C01827=1144.684,360.117,-81.640,-176.368,9.412,148.862
C01828=1144.680,360.365,-81.675,-176.367,9.416,148.862
C01829=1144.676,360.613,-81.711,-176.364,9.420,148.863
C01830=1144.671,360.859,-81.746,-176.361,9.425,148.863
C01831=1144.667,361.107,-81.781,-176.358,9.429,148.863
C01832=1144.664,361.355,-81.817,-176.356,9.432,148.864
C01833=1144.660,361.602,-81.852,-176.353,9.436,148.864
C01834=1144.656,361.849,-81.888,-176.351,9.441,148.865
C01835=1144.652,362.097,-81.923,-176.348,9.445,148.865
C01836=1144.648,362.344,-81.959,-176.345,9.449,148.865
C01837=1144.644,362.592,-81.993,-176.344,9.453,148.866
C01838=1144.640,362.839,-82.029,-176.341,9.457,148.866
C01839=1144.637,363.087,-82.064,-176.338,9.461,148.866
C01840=1144.633,363.334,-82.100,-176.335,9.465,148.867
C01841=1144.629,363.582,-82.135,-176.333,9.470,148.867
C01842=1144.626,363.829,-82.171,-176.330,9.474,148.867
C01843=1144.621,364.077,-82.207,-176.328,9.477,148.868
C01844=1144.617,364.324,-82.242,-176.325,9.481,148.868
C01845=1144.613,364.571,-82.278,-176.322,9.486,148.869
C01846=1144.609,364.855,-82.318,-176.319,9.491,148.869
C01847=1144.604,365.138,-82.359,-176.316,9.495,148.869
C01848=1144.601,365.422,-82.400,-176.313,9.500,148.870
C01849=1144.596,365.705,-82.441,-176.310,9.504,148.870
C01850=1144.592,365.953,-82.477,-176.308,9.508,148.870
C01851=1144.587,366.200,-82.513,-176.305,9.513,148.871
C01852=1144.584,366.448,-82.548,-176.303,9.517,148.871
C01853=1144.580,366.695,-82.584,-176.300,9.521,148.872
C01854=1144.576,366.943,-82.620,-176.297,9.526,148.872
C01855=1144.572,367.190,-82.656,-176.294,9.530,148.872
C01856=1144.569,367.437,-82.692,-176.292,9.534,148.873
C01857=1144.565,367.685,-82.727,-176.289,9.538,148.873
C01858=1144.561,367.933,-82.763,-176.287,9.542,148.874
C01859=1144.556,368.179,-82.798,-176.284,9.546,148.874
C01860=1144.553,368.426,-82.835,-176.281,9.550,148.874
C01861=1144.549,368.674,-82.871,-176.279,9.555,148.875
C01862=1144.545,368.922,-82.906,-176.276,9.559,148.875
C01863=1144.542,369.168,-82.943,-176.273,9.563,148.875
C01864=1144.537,369.416,-82.979,-176.271,9.567,148.876
C01865=1144.534,369.664,-83.014,-176.268,9.572,148.876
C01866=1144.530,369.911,-83.051,-176.266,9.576,148.877
C01867=1144.526,370.158,-83.087,-176.263,9.580,148.877
C01868=1144.522,370.406,-83.122,-176.260,9.584,148.877
C01869=1144.518,370.653,-83.159,-176.258,9.588,148.878
C01870=1144.514,370.901,-83.195,-176.256,9.592,148.878
C01871=1144.511,371.148,-83.231,-176.253,9.596,148.879
C01872=1144.507,371.395,-83.267,-176.250,9.601,148.879
C01873=1144.503,371.643,-83.303,-176.248,9.605,148.879
C01874=1144.499,371.890,-83.340,-176.245,9.610,148.880
C01875=1144.495,372.138,-83.375,-176.243,9.614,148.880
C01876=1144.491,372.385,-83.412,-176.240,9.618,148.881
C01877=1144.487,372.632,-83.447,-176.238,9.622,148.881
C01878=1144.483,372.879,-83.484,-176.235,9.626,148.882
C01879=1144.480,373.126,-83.521,-176.233,9.630,148.882
C01880=1144.476,373.374,-83.557,-176.230,9.635,148.883
C01881=1144.472,373.621,-83.593,-176.228,9.639,148.883
C01882=1144.468,373.869,-83.629,-176.226,9.643,148.883
C01883=1144.465,374.116,-83.665,-176.223,9.647,148.884
C01884=1144.460,374.363,-83.702,-176.221,9.652,148.884
C01885=1144.457,374.610,-83.738,-176.218,9.656,148.885
C01886=1144.453,374.858,-83.775,-176.217,9.659,148.885
C01887=1144.449,375.105,-83.810,-176.214,9.664,148.886
C01888=1144.445,375.352,-83.847,-176.212,9.668,148.886
C01889=1144.441,375.599,-83.884,-176.210,9.672,148.887
C01890=1144.438,375.847,-83.921,-176.207,9.676,148.887
C01891=1144.434,376.095,-83.957,-176.205,9.681,148.888
C01892=1144.430,376.342,-83.993,-176.203,9.684,148.888
C01893=1144.426,376.589,-84.030,-176.201,9.689,148.889
C01894=1144.422,376.836,-84.067,-176.199,9.692,148.889
C01895=1144.418,377.084,-84.102,-176.197,9.697,148.890
C01896=1144.414,377.331,-84.139,-176.195,9.701,148.890
C01897=1144.410,377.578,-84.176,-176.193,9.705,148.891
C01898=1144.407,377.825,-84.212,-176.191,9.709,148.891
C01899=1144.403,378.073,-84.249,-176.189,9.713,148.892
C01900=1144.399,378.321,-84.286,-176.187,9.717,148.892
C01901=1144.396,378.567,-84.322,-176.185,9.721,148.893
C01902=1144.392,378.815,-84.359,-176.183,9.725,148.893
C01903=1144.387,379.062,-84.396,-176.181,9.729,148.894
C01904=1144.383,379.309,-84.432,-176.179,9.733,148.894
C01905=1144.380,379.556,-84.469,-176.178,9.737,148.895
C01906=1144.377,379.804,-84.506,-176.176,9.741,148.896
C01907=1144.372,380.051,-84.543,-176.175,9.745,148.896
C01908=1144.369,380.298,-84.579,-176.173,9.749,148.897
C01909=1144.365,380.545,-84.616,-176.171,9.752,148.897
C01910=1144.361,380.792,-84.653,-176.170,9.756,148.898
C01911=1144.357,381.039,-84.690,-176.168,9.760,148.898
C01912=1144.354,381.287,-84.726,-176.167,9.764,148.899
C01913=1144.350,381.534,-84.763,-176.166,9.767,148.900
C01914=1144.346,381.781,-84.800,-176.165,9.771,148.900
C01915=1144.342,382.029,-84.837,-176.163,9.775,148.901
C01916=1144.338,382.276,-84.874,-176.162,9.779,148.902
C01917=1144.335,382.523,-84.910,-176.161,9.782,148.902
C01918=1144.331,382.771,-84.947,-176.160,9.786,148.903
C01919=1144.327,383.018,-84.984,-176.159,9.789,148.904
C01920=1144.323,383.265,-85.021,-176.158,9.792,148.904
C01921=1144.319,383.512,-85.058,-176.157,9.796,148.905
C01922=1144.315,383.760,-85.095,-176.156,9.799,148.906
C01923=1144.312,384.007,-85.131,-176.156,9.803,148.906
C01924=1144.308,384.254,-85.168,-176.155,9.806,148.907
C01925=1144.304,384.501,-85.206,-176.154,9.809,148.908
C01926=1144.300,384.749,-85.243,-176.154,9.813,148.908
C01927=1144.296,384.996,-85.280,-176.153,9.816,148.909
C01928=1144.292,385.243,-85.317,-176.153,9.819,148.910
C01929=1144.289,385.490,-85.353,-176.152,9.823,148.911
C01930=1144.285,385.738,-85.390,-176.152,9.825,148.911
C01931=1144.281,385.984,-85.428,-176.152,9.829,148.912
C01932=1144.277,386.231,-85.465,-176.151,9.832,148.913
C01933=1144.273,386.479,-85.501,-176.151,9.835,148.914
C01934=1144.270,386.727,-85.539,-176.151,9.838,148.914
C01935=1144.266,386.974,-85.575,-176.151,9.841,148.915
C01936=1144.262,387.221,-85.612,-176.152,9.843,148.916
C01937=1144.259,387.467,-85.649,-176.151,9.847,148.917
C01938=1144.255,387.715,-85.687,-176.151,9.849,148.917
C01939=1144.251,387.962,-85.723,-176.151,9.852,148.918
C01940=1144.247,388.209,-85.760,-176.152,9.855,148.919
C01941=1144.243,388.456,-85.798,-176.152,9.857,148.920
C01942=1144.240,388.704,-85.835,-176.152,9.860,148.921
C01943=1144.235,388.951,-85.872,-176.152,9.863,148.921
C01944=1144.231,389.198,-85.909,-176.153,9.866,148.922
C01945=1144.228,389.446,-85.946,-176.153,9.868,148.923
C01946=1144.224,389.693,-85.984,-176.154,9.871,148.924
C01947=1144.221,389.940,-86.020,-176.154,9.874,148.924
C01948=1144.217,390.187,-86.057,-176.155,9.876,148.925
C01949=1144.213,390.435,-86.094,-176.155,9.879,148.926
C01950=1144.208,390.721,-86.138,-176.156,9.881,148.927
C01951=1144.205,391.009,-86.180,-176.156,9.884,148.928
C01952=1144.200,391.295,-86.224,-176.157,9.888,148.929
C01953=1144.195,391.582,-86.266,-176.158,9.890,148.930
C01954=1144.192,391.830,-86.304,-176.159,9.892,148.931
C01955=1144.188,392.076,-86.341,-176.160,9.895,148.932
C01956=1144.184,392.324,-86.378,-176.160,9.897,148.932
C01957=1144.180,392.571,-86.415,-176.161,9.899,148.933
C01958=1144.176,392.819,-86.452,-176.162,9.902,148.934
C01959=1144.173,393.065,-86.490,-176.163,9.904,148.935
C01960=1144.168,393.312,-86.526,-176.164,9.906,148.936
C01961=1144.165,393.560,-86.564,-176.164,9.909,148.937
C01962=1144.162,393.807,-86.601,-176.165,9.911,148.937
C01963=1144.158,394.054,-86.638,-176.166,9.913,148.938
C01964=1144.154,394.302,-86.675,-176.167,9.915,148.939
C01965=1144.150,394.549,-86.712,-176.168,9.918,148.940
C01966=1144.146,394.795,-86.749,-176.169,9.920,148.941
C01967=1144.142,395.043,-86.786,-176.170,9.922,148.941
C01968=1144.139,395.290,-86.823,-176.171,9.924,148.942
C01969=1144.135,395.538,-86.860,-176.172,9.926,148.943
C01970=1144.131,395.784,-86.898,-176.173,9.928,148.944
C01971=1144.127,396.032,-86.935,-176.174,9.930,148.945
C01972=1144.123,396.279,-86.972,-176.175,9.932,148.946
C01973=1144.120,396.526,-87.009,-176.177,9.934,148.946
C01974=1144.115,396.773,-87.046,-176.178,9.936,148.947
C01975=1144.112,397.021,-87.083,-176.179,9.938,148.948
C01976=1144.108,397.268,-87.121,-176.180,9.940,148.949
C01977=1144.104,397.515,-87.158,-176.181,9.942,148.950
C01978=1144.101,397.763,-87.195,-176.182,9.945,148.951
C01979=1144.096,398.010,-87.232,-176.183,9.947,148.951
C01980=1144.093,398.256,-87.270,-176.184,9.949,148.952
C01981=1144.089,398.504,-87.306,-176.185,9.951,148.953
C01982=1144.086,398.751,-87.343,-176.186,9.953,148.954
C01983=1144.082,398.998,-87.381,-176.187,9.955,148.955
C01984=1144.078,399.245,-87.417,-176.189,9.957,148.956
C01985=1144.074,399.493,-87.455,-176.190,9.959,148.956
C01986=1144.070,399.740,-87.492,-176.191,9.961,148.957
C01987=1144.067,399.987,-87.529,-176.193,9.963,148.958
C01988=1144.062,400.234,-87.566,-176.194,9.965,148.959
C01989=1144.059,400.482,-87.603,-176.195,9.967,148.960
C01990=1144.055,400.728,-87.641,-176.196,9.969,148.961
C01991=1144.051,400.975,-87.678,-176.197,9.971,148.962
C01992=1144.048,401.223,-87.715,-176.198,9.973,148.962
C01993=1144.044,401.470,-87.752,-176.199,9.975,148.963
C01994=1144.040,401.717,-87.789,-176.201,9.976,148.964
C01995=1144.036,401.964,-87.826,-176.202,9.978,148.965
C01996=1144.032,402.212,-87.863,-176.203,9.980,148.966
C01997=1144.028,402.459,-87.901,-176.204,9.982,148.967
C01998=1144.024,402.706,-87.938,-176.205,9.984,148.967
C01999=1144.021,402.954,-87.975,-176.206,9.986,148.968
C02000=1144.017,403.201,-88.012,-176.208,9.987,148.969
C02001=1144.013,403.448,-88.049,-176.209,9.990,148.970
C02002=1144.010,403.695,-88.086,-176.210,9.992,148.970
C02003=1144.006,403.942,-88.123,-176.211,9.994,148.971
C02004=1144.002,404.189,-88.161,-176.212,9.996,148.972
C02005=1143.998,404.436,-88.197,-176.213,9.998,148.973
C02006=1143.995,404.684,-88.235,-176.214,10.000,148.974
C02007=1143.991,404.931,-88.271,-176.216,10.001,148.975
C02008=1143.987,405.178,-88.309,-176.217,10.003,148.975
C02009=1143.983,405.426,-88.346,-176.218,10.005,148.976
C02010=1143.979,405.673,-88.383,-176.219,10.007,148.977
C02011=1143.975,405.919,-88.421,-176.220,10.009,148.978
C02012=1143.971,406.167,-88.458,-176.221,10.011,148.978
C02013=1143.968,406.414,-88.495,-176.222,10.013,148.979
C02014=1143.964,406.661,-88.532,-176.223,10.015,148.980
C02015=1143.960,406.908,-88.569,-176.224,10.017,148.981
C02016=1143.956,407.156,-88.606,-176.226,10.019,148.982
C02017=1143.952,407.403,-88.643,-176.227,10.021,148.983
C02018=1143.949,407.650,-88.681,-176.228,10.022,148.983
C02019=1143.944,407.897,-88.718,-176.229,10.024,148.984
C02020=1143.941,408.145,-88.755,-176.230,10.027,148.985
C02021=1143.938,408.391,-88.792,-176.231,10.029,148.986
C02022=1143.934,408.638,-88.829,-176.232,10.030,148.986
C02023=1143.930,408.886,-88.866,-176.233,10.032,148.987
C02024=1143.926,409.133,-88.903,-176.234,10.034,148.988
C02025=1143.922,409.380,-88.940,-176.235,10.037,148.989
C02026=1143.918,409.627,-88.977,-176.236,10.038,148.989
C02027=1143.915,409.875,-89.015,-176.237,10.040,148.990
C02028=1143.911,410.122,-89.052,-176.238,10.042,148.991
C02029=1143.907,410.369,-89.089,-176.239,10.044,148.992
C02030=1143.903,410.617,-89.126,-176.239,10.046,148.993
C02031=1143.899,410.864,-89.163,-176.241,10.048,148.993
C02032=1143.896,411.111,-89.201,-176.242,10.050,148.994
C02033=1143.892,411.358,-89.237,-176.242,10.052,148.995
C02034=1143.888,411.606,-89.275,-176.243,10.054,148.996
C02035=1143.884,411.852,-89.312,-176.243,10.057,148.996
C02036=1143.880,412.099,-89.349,-176.245,10.059,148.997
C02037=1143.877,412.347,-89.386,-176.246,10.061,148.998
C02038=1143.873,412.594,-89.424,-176.246,10.063,148.999
C02039=1143.869,412.841,-89.461,-176.247,10.065,149.000
C02040=1143.865,413.088,-89.498,-176.248,10.066,149.000
C02041=1143.861,413.336,-89.535,-176.249,10.069,149.001
C02042=1143.857,413.583,-89.572,-176.250,10.071,149.002
C02043=1143.853,413.830,-89.609,-176.250,10.073,149.003
C02044=1143.850,414.078,-89.647,-176.251,10.075,149.003
C02045=1143.846,414.324,-89.684,-176.252,10.077,149.004
C02046=1143.843,414.571,-89.720,-176.253,10.079,149.005
C02047=1143.839,414.819,-89.758,-176.254,10.081,149.005
C02048=1143.837,415.066,-89.795,-176.254,10.084,149.006
C02049=1143.835,415.313,-89.832,-176.255,10.085,149.007
C02050=1143.834,415.560,-89.869,-176.256,10.087,149.008
C02051=1143.833,415.808,-89.906,-176.257,10.089,149.008
C02052=1143.834,416.055,-89.942,-176.257,10.091,149.009
C02053=1143.835,416.302,-89.978,-176.258,10.094,149.010
C02054=1143.836,416.549,-90.016,-176.258,10.096,149.011
C02055=1143.839,416.796,-90.052,-176.259,10.097,149.011
C02056=1143.842,417.043,-90.088,-176.260,10.099,149.012
C02057=1143.845,417.289,-90.124,-176.260,10.101,149.013
C02058=1143.425,417.292,-90.174,-176.262,10.112,149.016
C02059=1143.421,417.042,-90.138,-176.262,10.111,149.015
C02060=1143.418,416.791,-90.101,-176.261,10.109,149.015
C02061=1143.416,416.541,-90.064,-176.261,10.106,149.014
C02062=1143.414,416.290,-90.027,-176.260,10.104,149.013
C02063=1143.413,416.043,-89.990,-176.259,10.102,149.013
C02064=1143.413,415.796,-89.954,-176.258,10.100,149.012
C02065=1143.413,415.549,-89.917,-176.258,10.099,149.011
C02066=1143.415,415.302,-89.880,-176.257,10.096,149.010
C02067=1143.416,415.054,-89.843,-176.256,10.094,149.010
C02068=1143.418,414.807,-89.806,-176.256,10.092,149.009
C02069=1143.422,414.560,-89.769,-176.255,10.090,149.008
C02070=1143.426,414.312,-89.731,-176.254,10.088,149.007
C02071=1143.430,414.065,-89.694,-176.253,10.086,149.007
C02072=1143.434,413.819,-89.657,-176.252,10.084,149.006
C02073=1143.437,413.571,-89.620,-176.252,10.082,149.005
C02074=1143.441,413.324,-89.583,-176.251,10.080,149.004
C02075=1143.445,413.077,-89.545,-176.250,10.078,149.004
C02076=1143.449,412.830,-89.508,-176.249,10.076,149.003
C02077=1143.453,412.582,-89.471,-176.248,10.073,149.002
C02078=1143.456,412.335,-89.434,-176.248,10.071,149.001
C02079=1143.460,412.088,-89.397,-176.247,10.069,149.001
C02080=1143.464,411.840,-89.360,-176.246,10.067,149.000
C02081=1143.467,411.594,-89.323,-176.245,10.065,148.999
C02082=1143.471,411.347,-89.286,-176.244,10.063,148.998
C02083=1143.475,411.099,-89.248,-176.243,10.061,148.997
C02084=1143.479,410.852,-89.212,-176.242,10.059,148.997
C02085=1143.482,410.605,-89.174,-176.241,10.057,148.996
C02086=1143.487,410.358,-89.137,-176.240,10.055,148.995
C02087=1143.490,410.110,-89.100,-176.239,10.054,148.994
C02088=1143.494,409.863,-89.062,-176.238,10.052,148.994
C02089=1143.498,409.616,-89.025,-176.237,10.049,148.993
C02090=1143.501,409.368,-88.988,-176.236,10.047,148.992
C02091=1143.505,409.122,-88.951,-176.235,10.046,148.991
C02092=1143.509,408.875,-88.914,-176.234,10.044,148.991
C02093=1143.513,408.627,-88.877,-176.233,10.042,148.990
C02094=1143.517,408.380,-88.839,-176.232,10.039,148.989
C02095=1143.521,408.133,-88.802,-176.231,10.037,148.988
C02096=1143.525,407.886,-88.765,-176.230,10.036,148.987
C02097=1143.528,407.638,-88.728,-176.229,10.034,148.987
C02098=1143.532,407.391,-88.691,-176.228,10.032,148.986
C02099=1143.536,407.144,-88.654,-176.227,10.029,148.985
C02100=1143.540,406.896,-88.616,-176.226,10.027,148.984
C02101=1143.543,406.650,-88.579,-176.225,10.025,148.983
C02102=1143.548,406.402,-88.542,-176.224,10.023,148.982
C02103=1143.552,406.155,-88.505,-176.223,10.022,148.982
C02104=1143.555,405.908,-88.467,-176.222,10.019,148.981
C02105=1143.559,405.661,-88.430,-176.221,10.017,148.980
C02106=1143.562,405.414,-88.394,-176.219,10.016,148.979
C02107=1143.565,405.167,-88.356,-176.218,10.014,148.979
C02108=1143.570,404.919,-88.319,-176.217,10.012,148.978
C02109=1143.574,404.672,-88.282,-176.216,10.010,148.977
C02110=1143.578,404.425,-88.246,-176.215,10.008,148.976
C02111=1143.581,404.178,-88.208,-176.214,10.006,148.975
C02112=1143.585,403.931,-88.171,-176.213,10.004,148.974
C02113=1143.589,403.683,-88.134,-176.211,10.002,148.974
C02114=1143.592,403.436,-88.096,-176.210,10.000,148.973
C02115=1143.596,403.189,-88.059,-176.209,9.998,148.972
C02116=1143.600,402.942,-88.022,-176.208,9.996,148.971
C02117=1143.604,402.695,-87.984,-176.207,9.994,148.970
C02118=1143.608,402.447,-87.947,-176.206,9.992,148.969
C02119=1143.612,402.200,-87.911,-176.204,9.991,148.969
C02120=1143.616,401.953,-87.874,-176.203,9.989,148.968
C02121=1143.619,401.706,-87.836,-176.202,9.987,148.967
C02122=1143.623,401.459,-87.799,-176.201,9.985,148.966
C02123=1143.627,401.211,-87.762,-176.200,9.983,148.965
C02124=1143.631,400.964,-87.724,-176.199,9.981,148.964
C02125=1143.635,400.717,-87.687,-176.197,9.979,148.964
C02126=1143.639,400.470,-87.650,-176.196,9.977,148.963
C02127=1143.643,400.223,-87.613,-176.195,9.975,148.962
C02128=1143.646,399.975,-87.576,-176.194,9.973,148.961
C02129=1143.649,399.728,-87.539,-176.192,9.971,148.960
C02130=1143.653,399.482,-87.502,-176.191,9.969,148.960
C02131=1143.657,399.234,-87.465,-176.190,9.967,148.959
C02132=1143.661,398.987,-87.428,-176.189,9.965,148.958
C02133=1143.665,398.739,-87.391,-176.188,9.963,148.957
C02134=1143.668,398.492,-87.353,-176.186,9.962,148.956
C02135=1143.672,398.245,-87.316,-176.185,9.960,148.955
C02136=1143.676,397.998,-87.279,-176.184,9.957,148.955
C02137=1143.680,397.751,-87.242,-176.183,9.955,148.954
C02138=1143.683,397.503,-87.204,-176.182,9.953,148.953
C02139=1143.688,397.256,-87.168,-176.181,9.951,148.952
C02140=1143.691,397.010,-87.130,-176.180,9.949,148.951
C02141=1143.695,396.762,-87.093,-176.179,9.947,148.950
C02142=1143.699,396.515,-87.056,-176.178,9.945,148.950
C02143=1143.703,396.267,-87.019,-176.177,9.943,148.949
C02144=1143.707,396.021,-86.981,-176.175,9.941,148.948
C02145=1143.710,395.773,-86.944,-176.174,9.939,148.947
C02146=1143.714,395.526,-86.907,-176.173,9.937,148.946
C02147=1143.718,395.279,-86.870,-176.172,9.935,148.945
C02148=1143.722,395.031,-86.833,-176.172,9.932,148.945
C02149=1143.726,394.784,-86.796,-176.171,9.930,148.944
C02150=1143.730,394.537,-86.758,-176.170,9.928,148.943
C02151=1143.734,394.290,-86.721,-176.168,9.926,148.942
C02152=1143.737,394.042,-86.684,-176.167,9.924,148.941
C02153=1143.741,393.796,-86.648,-176.167,9.921,148.940
C02154=1143.744,393.549,-86.610,-176.166,9.919,148.939
C02155=1143.748,393.301,-86.573,-176.165,9.917,148.939
C02156=1143.752,393.054,-86.536,-176.164,9.915,148.938
C02157=1143.756,392.807,-86.499,-176.163,9.912,148.937
C02158=1143.759,392.559,-86.461,-176.162,9.910,148.936
C02159=1143.763,392.312,-86.424,-176.161,9.908,148.935
C02160=1143.767,392.065,-86.388,-176.161,9.905,148.935
C02161=1143.771,391.818,-86.350,-176.160,9.903,148.934
C02162=1143.775,391.571,-86.313,-176.160,9.900,148.933
C02163=1143.779,391.284,-86.270,-176.159,9.897,148.932
C02164=1143.783,390.997,-86.226,-176.158,9.895,148.931
C02165=1143.788,390.710,-86.184,-176.157,9.892,148.930
C02166=1143.792,390.423,-86.140,-176.156,9.889,148.929
C02167=1143.796,390.175,-86.103,-176.156,9.887,148.928
C02168=1143.800,389.928,-86.066,-176.155,9.884,148.928
C02169=1143.804,389.681,-86.029,-176.155,9.881,148.927
C02170=1143.807,389.434,-85.992,-176.154,9.879,148.926
C02171=1143.811,389.187,-85.955,-176.154,9.877,148.925
C02172=1143.815,388.940,-85.918,-176.154,9.874,148.924
C02173=1143.818,388.692,-85.881,-176.154,9.871,148.924
C02174=1143.822,388.445,-85.844,-176.153,9.868,148.923
C02175=1143.826,388.198,-85.807,-176.153,9.866,148.922
C02176=1143.830,387.951,-85.770,-176.152,9.863,148.921
C02177=1143.834,387.703,-85.733,-176.152,9.860,148.921
C02178=1143.838,387.456,-85.695,-176.153,9.857,148.920
C02179=1143.842,387.209,-85.658,-176.153,9.854,148.919
C02180=1143.846,386.962,-85.621,-176.152,9.851,148.918
C02181=1143.849,386.714,-85.585,-176.153,9.848,148.917
C02182=1143.853,386.467,-85.548,-176.153,9.845,148.917
C02183=1143.856,386.221,-85.510,-176.153,9.842,148.916
C02184=1143.860,385.973,-85.473,-176.153,9.840,148.915
C02185=1143.864,385.726,-85.436,-176.154,9.836,148.915
C02186=1143.868,385.478,-85.399,-176.153,9.834,148.914
C02187=1143.872,385.231,-85.363,-176.154,9.830,148.913
C02188=1143.875,384.984,-85.325,-176.154,9.827,148.912
C02189=1143.879,384.737,-85.288,-176.155,9.824,148.912
C02190=1143.883,384.490,-85.251,-176.156,9.820,148.911
C02191=1143.887,384.243,-85.215,-176.156,9.817,148.910
C02192=1143.890,383.995,-85.177,-176.157,9.814,148.910
C02193=1143.895,383.748,-85.141,-176.158,9.811,148.909
C02194=1143.899,383.500,-85.104,-176.159,9.808,148.908
C02195=1143.903,383.253,-85.067,-176.160,9.803,148.908
C02196=1143.906,383.007,-85.030,-176.161,9.800,148.907
C02197=1143.909,382.759,-84.993,-176.162,9.796,148.906
C02198=1143.913,382.512,-84.956,-176.163,9.793,148.906
C02199=1143.917,382.265,-84.919,-176.164,9.789,148.905
C02200=1143.922,382.018,-84.882,-176.165,9.786,148.904
C02201=1143.924,381.770,-84.845,-176.166,9.782,148.904
C02202=1143.928,381.523,-84.809,-176.168,9.778,148.903
C02203=1143.933,381.276,-84.772,-176.169,9.775,148.902
C02204=1143.937,381.028,-84.735,-176.170,9.771,148.902
C02205=1143.941,380.781,-84.698,-176.172,9.767,148.901
C02206=1143.944,380.534,-84.662,-176.173,9.763,148.901
C02207=1143.948,380.286,-84.624,-176.175,9.760,148.900
C02208=1143.952,380.039,-84.588,-176.176,9.756,148.900
C02209=1143.956,379.792,-84.551,-176.178,9.752,148.899
C02210=1143.959,379.545,-84.515,-176.179,9.748,148.898
C02211=1143.963,379.298,-84.478,-176.181,9.744,148.898
C02212=1143.967,379.050,-84.440,-176.183,9.740,148.897
C02213=1143.970,378.803,-84.404,-176.185,9.736,148.897
C02214=1143.974,378.555,-84.368,-176.187,9.732,148.896
C02215=1143.979,378.308,-84.331,-176.188,9.728,148.896
C02216=1143.983,378.061,-84.294,-176.191,9.724,148.895
C02217=1143.986,377.814,-84.258,-176.192,9.720,148.895
C02218=1143.990,377.567,-84.221,-176.195,9.716,148.894
C02219=1143.994,377.320,-84.184,-176.197,9.712,148.894
C02220=1143.997,377.072,-84.148,-176.198,9.708,148.893
C02221=1144.001,376.824,-84.112,-176.201,9.704,148.893
C02222=1144.005,376.577,-84.075,-176.203,9.700,148.892
C02223=1144.009,376.330,-84.038,-176.205,9.696,148.892
C02224=1144.013,376.083,-84.002,-176.207,9.691,148.891
C02225=1144.017,375.836,-83.966,-176.209,9.688,148.891
C02226=1144.021,375.588,-83.929,-176.212,9.683,148.890
C02227=1144.025,375.341,-83.892,-176.214,9.679,148.890
C02228=1144.028,375.094,-83.856,-176.216,9.675,148.889
C02229=1144.032,374.847,-83.820,-176.219,9.671,148.889
C02230=1144.036,374.600,-83.784,-176.221,9.667,148.888
C02231=1144.039,374.352,-83.746,-176.223,9.663,148.888
C02232=1144.043,374.104,-83.711,-176.225,9.658,148.887
C02233=1144.047,373.857,-83.674,-176.228,9.654,148.887
C02234=1144.051,373.609,-83.638,-176.231,9.650,148.887
C02235=1144.055,373.362,-83.602,-176.233,9.646,148.886
C02236=1144.059,373.115,-83.565,-176.235,9.642,148.886
C02237=1144.063,372.868,-83.529,-176.238,9.638,148.885
C02238=1144.067,372.620,-83.492,-176.240,9.633,148.885
C02239=1144.070,372.373,-83.457,-176.243,9.629,148.884
C02240=1144.074,372.126,-83.420,-176.245,9.624,148.884
C02241=1144.078,371.878,-83.384,-176.247,9.621,148.884
C02242=1144.081,371.631,-83.348,-176.250,9.617,148.883
C02243=1144.086,371.384,-83.312,-176.252,9.612,148.883
C02244=1144.089,371.137,-83.276,-176.255,9.608,148.882
C02245=1144.094,370.889,-83.240,-176.258,9.604,148.882
C02246=1144.097,370.642,-83.203,-176.260,9.599,148.881
C02247=1144.101,370.394,-83.167,-176.263,9.595,148.881
C02248=1144.105,370.147,-83.132,-176.265,9.591,148.880
C02249=1144.108,369.900,-83.095,-176.268,9.587,148.880
C02250=1144.113,369.652,-83.059,-176.271,9.582,148.880
C02251=1144.116,369.405,-83.024,-176.273,9.579,148.879
C02252=1144.121,369.157,-82.987,-176.276,9.575,148.879
C02253=1144.124,368.910,-82.951,-176.278,9.570,148.879
C02254=1144.128,368.662,-82.916,-176.281,9.566,148.878
C02255=1144.133,368.416,-82.879,-176.284,9.562,148.878
C02256=1144.136,368.168,-82.844,-176.286,9.557,148.877
C02257=1144.140,367.921,-82.808,-176.289,9.553,148.877
C02258=1144.144,367.673,-82.772,-176.291,9.549,148.877
C02259=1144.148,367.426,-82.736,-176.294,9.545,148.876
C02260=1144.151,367.179,-82.700,-176.297,9.540,148.876
C02261=1144.155,366.931,-82.665,-176.299,9.536,148.875
C02262=1144.159,366.683,-82.628,-176.302,9.532,148.875
C02263=1144.163,366.436,-82.593,-176.304,9.528,148.875
C02264=1144.167,366.189,-82.558,-176.307,9.524,148.875
C02265=1144.171,365.942,-82.521,-176.310,9.520,148.874
C02266=1144.175,365.694,-82.485,-176.313,9.516,148.874
C02267=1144.179,365.411,-82.445,-176.316,9.511,148.873
C02268=1144.183,365.127,-82.403,-176.318,9.506,148.873
C02269=1144.188,364.844,-82.363,-176.322,9.501,148.872
C02270=1144.192,364.560,-82.322,-176.325,9.496,148.872
C02271=1144.196,364.313,-82.286,-176.327,9.493,148.872
C02272=1144.200,364.066,-82.251,-176.330,9.489,148.871
C02273=1144.204,363.818,-82.215,-176.333,9.484,148.871
C02274=1144.208,363.571,-82.179,-176.335,9.480,148.871
C02275=1144.212,363.322,-82.145,-176.338,9.476,148.870
C02276=1144.216,363.075,-82.109,-176.340,9.472,148.870
C02277=1144.219,362.827,-82.073,-176.343,9.468,148.870
C02278=1144.224,362.581,-82.038,-176.345,9.464,148.869
C02279=1144.227,362.333,-82.003,-176.348,9.460,148.869
C02280=1144.231,362.086,-81.967,-176.351,9.455,148.868
C02281=1144.235,361.838,-81.932,-176.354,9.451,148.868
C02282=1144.239,361.591,-81.896,-176.356,9.448,148.868
C02283=1144.243,361.344,-81.860,-176.358,9.443,148.867
C02284=1144.247,361.095,-81.826,-176.361,9.439,148.867
C02285=1144.251,360.848,-81.790,-176.363,9.435,148.867
C02286=1144.255,360.600,-81.754,-176.366,9.431,148.866
C02287=1144.259,360.354,-81.719,-176.368,9.427,148.866
C02288=1144.263,360.106,-81.684,-176.371,9.423,148.866
C02289=1144.267,359.858,-81.649,-176.374,9.419,148.865
C02290=1144.271,359.611,-81.614,-176.377,9.415,148.865
C02291=1144.274,359.364,-81.578,-176.379,9.411,148.865
C02292=1144.278,359.116,-81.543,-176.382,9.407,148.864
C02293=1144.282,358.868,-81.508,-176.384,9.403,148.864
C02294=1144.286,358.621,-81.473,-176.386,9.399,148.864
C02295=1144.290,358.373,-81.438,-176.389,9.395,148.863
C02296=1144.293,358.126,-81.403,-176.392,9.391,148.863
C02297=1144.298,357.879,-81.368,-176.394,9.387,148.862
C02298=1144.301,357.631,-81.333,-176.397,9.383,148.862
C02299=1144.305,357.384,-81.297,-176.399,9.379,148.862
C02300=1144.309,357.137,-81.262,-176.402,9.375,148.861
C02301=1144.313,356.889,-81.227,-176.404,9.371,148.861
C02302=1144.317,356.641,-81.192,-176.407,9.367,148.861
C02303=1144.322,356.394,-81.157,-176.409,9.363,148.860
C02304=1144.325,356.146,-81.122,-176.412,9.360,148.860
C02305=1144.329,355.898,-81.087,-176.414,9.355,148.860
C02306=1144.333,355.652,-81.052,-176.417,9.351,148.859
C02307=1144.337,355.403,-81.017,-176.419,9.347,148.859
C02308=1144.340,355.156,-80.982,-176.422,9.343,148.859
C02309=1144.345,354.909,-80.947,-176.424,9.339,148.858
C02310=1144.349,354.660,-80.913,-176.427,9.336,148.858
C02311=1144.352,354.414,-80.878,-176.429,9.331,148.858
C02312=1144.356,354.166,-80.843,-176.432,9.327,148.857
C02313=1144.360,353.918,-80.808,-176.434,9.324,148.857
C02314=1144.365,353.671,-80.773,-176.437,9.320,148.857
C02315=1144.369,353.423,-80.738,-176.440,9.315,148.856
C02316=1144.372,353.176,-80.704,-176.442,9.312,148.856
C02317=1144.376,352.928,-80.669,-176.444,9.308,148.856
C02318=1144.381,352.681,-80.634,-176.447,9.303,148.855
C02319=1144.384,352.433,-80.599,-176.449,9.300,148.855
C02320=1144.388,352.185,-80.565,-176.452,9.296,148.855
C02321=1144.392,351.938,-80.530,-176.454,9.292,148.854
C02322=1144.396,351.690,-80.495,-176.457,9.288,148.854
C02323=1144.400,351.443,-80.461,-176.460,9.284,148.854
C02324=1144.404,351.195,-80.426,-176.462,9.281,148.853
C02325=1144.408,350.948,-80.391,-176.465,9.276,148.853
C02326=1144.412,350.700,-80.357,-176.467,9.272,148.853
C02327=1144.416,350.453,-80.323,-176.469,9.269,148.852
C02328=1144.420,350.205,-80.287,-176.472,9.264,148.852
C02329=1144.423,349.958,-80.253,-176.475,9.260,148.852
C02330=1144.427,349.710,-80.218,-176.477,9.257,148.852
C02331=1144.432,349.462,-80.184,-176.480,9.253,148.851
C02332=1144.435,349.215,-80.150,-176.482,9.249,148.851
C02333=1144.440,348.967,-80.115,-176.485,9.245,148.850
C02334=1144.444,348.719,-80.080,-176.487,9.241,148.850
C02335=1144.448,348.472,-80.047,-176.490,9.238,148.850
C02336=1144.452,348.224,-80.012,-176.492,9.233,148.849
C02337=1144.455,347.977,-79.978,-176.495,9.229,148.849
C02338=1144.460,347.729,-79.943,-176.497,9.226,148.849
C02339=1144.464,347.481,-79.909,-176.500,9.222,148.849
C02340=1144.468,347.234,-79.875,-176.502,9.218,148.848
C02341=1144.472,346.986,-79.840,-176.505,9.214,148.848
C02342=1144.476,346.739,-79.806,-176.508,9.210,148.848
C02343=1144.480,346.491,-79.771,-176.510,9.206,148.847
C02344=1144.483,346.244,-79.737,-176.513,9.202,148.847
C02345=1144.488,345.996,-79.703,-176.515,9.199,148.847
C02346=1144.491,345.748,-79.669,-176.517,9.194,148.846
C02347=1144.496,345.501,-79.634,-176.520,9.190,148.846
C02348=1144.499,345.253,-79.600,-176.523,9.187,148.846
C02349=1144.504,345.005,-79.566,-176.525,9.183,148.845
C02350=1144.508,344.758,-79.532,-176.528,9.179,148.845
C02351=1144.512,344.510,-79.497,-176.530,9.175,148.845
C02352=1144.516,344.263,-79.464,-176.533,9.171,148.845
C02353=1144.519,344.016,-79.430,-176.535,9.168,148.844
C02354=1144.524,343.767,-79.396,-176.538,9.164,148.844
C02355=1144.527,343.520,-79.362,-176.540,9.160,148.844
C02356=1144.531,343.272,-79.327,-176.543,9.156,148.843
C02357=1144.535,343.025,-79.293,-176.545,9.153,148.843
C02358=1144.540,342.777,-79.259,-176.548,9.148,148.843
C02359=1144.543,342.529,-79.225,-176.551,9.144,148.843
C02360=1144.547,342.282,-79.191,-176.553,9.141,148.842
C02361=1144.552,342.034,-79.157,-176.556,9.137,148.842
C02362=1144.556,341.787,-79.124,-176.558,9.133,148.842
C02363=1144.559,341.539,-79.089,-176.561,9.129,148.841
C02364=1144.564,341.291,-79.056,-176.563,9.126,148.841
C02365=1144.568,341.044,-79.022,-176.566,9.122,148.841
C02366=1144.571,340.795,-78.988,-176.569,9.117,148.841
C02367=1144.576,340.548,-78.954,-176.571,9.114,148.840
C02368=1144.580,340.300,-78.921,-176.573,9.110,148.840
C02369=1144.584,340.053,-78.887,-176.576,9.107,148.840
C02370=1144.588,339.805,-78.852,-176.579,9.102,148.839
C02371=1144.592,339.524,-78.814,-176.581,9.098,148.839
C02372=1144.597,339.245,-78.776,-176.584,9.094,148.839
C02373=1144.602,338.963,-78.738,-176.587,9.090,148.839
C02374=1144.606,338.683,-78.700,-176.590,9.086,148.838
C02375=1144.610,338.436,-78.666,-176.592,9.081,148.838
C02376=1144.614,338.187,-78.632,-176.595,9.077,148.838
C02377=1144.618,337.940,-78.598,-176.598,9.074,148.837
C02378=1144.622,337.692,-78.565,-176.601,9.070,148.837
C02379=1144.626,337.445,-78.531,-176.602,9.066,148.837
C02380=1144.630,337.197,-78.498,-176.605,9.062,148.837
C02381=1144.635,336.949,-78.464,-176.608,9.059,148.836
C02382=1144.638,336.702,-78.430,-176.611,9.055,148.836
C02383=1144.643,336.454,-78.397,-176.613,9.051,148.836
C02384=1144.647,336.206,-78.364,-176.615,9.047,148.835
C02385=1144.650,335.958,-78.330,-176.618,9.044,148.835
C02386=1144.654,335.711,-78.296,-176.621,9.040,148.835
C02387=1144.658,335.463,-78.263,-176.623,9.037,148.835
C02388=1144.662,335.215,-78.230,-176.626,9.032,148.834
C02389=1144.667,334.968,-78.196,-176.628,9.028,148.834
C02390=1144.671,334.720,-78.162,-176.631,9.025,148.834
C02391=1144.675,334.472,-78.129,-176.634,9.021,148.834
C02392=1144.679,334.224,-78.096,-176.636,9.018,148.833
C02393=1144.683,333.977,-78.062,-176.639,9.013,148.833
C02394=1144.687,333.729,-78.029,-176.641,9.010,148.833
C02395=1144.691,333.481,-77.996,-176.644,9.006,148.833
C02396=1144.695,333.234,-77.962,-176.646,9.003,148.832
C02397=1144.699,332.986,-77.929,-176.649,8.999,148.832
C02398=1144.703,332.737,-77.896,-176.651,8.995,148.832
C02399=1144.707,332.490,-77.863,-176.654,8.991,148.832
C02400=1144.711,332.242,-77.829,-176.656,8.988,148.831
C02401=1144.715,331.994,-77.796,-176.659,8.984,148.831
C02402=1144.719,331.747,-77.762,-176.661,8.980,148.831
C02403=1144.723,331.499,-77.729,-176.664,8.976,148.831
C02404=1144.727,331.252,-77.696,-176.667,8.973,148.830
C02405=1144.731,331.004,-77.663,-176.670,8.969,148.830
C02406=1144.735,330.756,-77.630,-176.671,8.965,148.830
C02407=1144.740,330.508,-77.597,-176.674,8.961,148.830
C02408=1144.744,330.261,-77.563,-176.677,8.958,148.829
C02409=1144.748,330.013,-77.530,-176.680,8.954,148.829
C02410=1144.752,329.765,-77.498,-176.682,8.951,148.829
C02411=1144.755,329.517,-77.465,-176.685,8.947,148.829
C02412=1144.759,329.269,-77.432,-176.687,8.943,148.829
C02413=1144.763,329.021,-77.399,-176.690,8.939,148.828
C02414=1144.768,328.773,-77.365,-176.692,8.936,148.828
C02415=1144.772,328.526,-77.332,-176.695,8.932,148.828
C02416=1144.776,328.278,-77.299,-176.697,8.928,148.827
C02417=1144.780,328.030,-77.266,-176.700,8.924,148.827
C02418=1144.784,327.782,-77.234,-176.703,8.921,148.827
C02419=1144.788,327.534,-77.201,-176.705,8.918,148.827
C02420=1144.792,327.287,-77.168,-176.708,8.914,148.827
C02421=1144.796,327.039,-77.135,-176.710,8.910,148.826
C02422=1144.800,326.791,-77.102,-176.713,8.906,148.826
C02423=1144.804,326.543,-77.070,-176.715,8.903,148.826
C02424=1144.808,326.295,-77.037,-176.718,8.899,148.826
C02425=1144.812,326.048,-77.003,-176.721,8.896,148.826
C02426=1144.817,325.799,-76.971,-176.724,8.892,148.825
C02427=1144.821,325.553,-76.939,-176.726,8.888,148.825
C02428=1144.825,325.305,-76.906,-176.729,8.884,148.825
C02429=1144.829,325.057,-76.872,-176.731,8.881,148.825
C02430=1144.833,324.809,-76.840,-176.734,8.877,148.824
C02431=1144.837,324.561,-76.807,-176.736,8.874,148.824
C02432=1144.841,324.313,-76.775,-176.739,8.870,148.824
C02433=1144.845,324.065,-76.742,-176.742,8.866,148.824
C02434=1144.849,323.818,-76.709,-176.744,8.863,148.823
C02435=1144.853,323.570,-76.677,-176.746,8.859,148.823
C02436=1144.857,323.322,-76.644,-176.749,8.855,148.823
C02437=1144.861,323.074,-76.612,-176.752,8.851,148.823
C02438=1144.865,322.826,-76.579,-176.754,8.848,148.823
C02439=1144.870,322.578,-76.546,-176.757,8.844,148.822
C02440=1144.874,322.331,-76.514,-176.759,8.841,148.822
C02441=1144.878,322.083,-76.482,-176.762,8.837,148.822
C02442=1144.881,321.835,-76.449,-176.765,8.833,148.822
C02443=1144.886,321.587,-76.417,-176.767,8.830,148.822
C02444=1144.890,321.339,-76.383,-176.770,8.826,148.822
C02445=1144.894,321.091,-76.352,-176.773,8.823,148.821
C02446=1144.898,320.843,-76.318,-176.775,8.819,148.821
C02447=1144.902,320.595,-76.287,-176.778,8.816,148.821
C02448=1144.907,320.348,-76.255,-176.780,8.812,148.821
C02449=1144.910,320.100,-76.222,-176.783,8.808,148.821
C02450=1144.914,319.852,-76.190,-176.785,8.805,148.820
C02451=1144.918,319.604,-76.158,-176.788,8.801,148.820
C02452=1144.922,319.356,-76.125,-176.791,8.798,148.820
C02453=1144.926,319.108,-76.093,-176.794,8.794,148.820
C02454=1144.931,318.861,-76.061,-176.796,8.790,148.820
C02455=1144.934,318.613,-76.028,-176.798,8.787,148.819
C02456=1144.939,318.365,-75.996,-176.801,8.783,148.819
C02457=1144.943,318.117,-75.964,-176.803,8.780,148.819
C02458=1144.947,317.869,-75.931,-176.806,8.776,148.819
C02459=1144.951,317.622,-75.899,-176.809,8.772,148.819
C02460=1144.955,317.373,-75.867,-176.811,8.769,148.818
C02461=1144.959,317.125,-75.835,-176.814,8.765,148.818
C02462=1144.964,316.877,-75.802,-176.817,8.762,148.818
C02463=1144.968,316.630,-75.770,-176.820,8.758,148.818
C02464=1144.971,316.382,-75.738,-176.822,8.755,148.818
C02465=1144.976,316.134,-75.706,-176.824,8.751,148.818
C02466=1144.980,315.886,-75.674,-176.827,8.747,148.817
C02467=1144.985,315.638,-75.642,-176.830,8.744,148.817
C02468=1144.988,315.390,-75.610,-176.832,8.740,148.817
C02469=1144.992,315.142,-75.578,-176.835,8.737,148.817
C02470=1144.996,314.894,-75.546,-176.837,8.734,148.817
C02471=1145.001,314.646,-75.514,-176.840,8.730,148.816
C02472=1145.004,314.398,-75.483,-176.843,8.726,148.816
C02473=1145.009,314.150,-75.450,-176.846,8.722,148.816
C02474=1145.013,313.903,-75.419,-176.848,8.719,148.816
C02475=1145.017,313.625,-75.383,-176.851,8.715,148.816
C02476=1145.023,313.347,-75.347,-176.854,8.711,148.815
C02477=1145.027,313.070,-75.311,-176.857,8.707,148.815
C02478=1145.032,312.792,-75.275,-176.860,8.703,148.815
C02479=1145.036,312.544,-75.243,-176.862,8.700,148.815
C02480=1145.039,312.296,-75.211,-176.865,8.697,148.815
C02481=1145.044,312.048,-75.180,-176.868,8.693,148.815
C02482=1145.048,311.800,-75.147,-176.870,8.689,148.814
C02483=1145.052,311.551,-75.116,-176.873,8.686,148.814
C02484=1145.056,311.304,-75.085,-176.876,8.682,148.814
C02485=1145.060,311.056,-75.053,-176.878,8.679,148.814
C02486=1145.064,310.808,-75.021,-176.880,8.676,148.814
C02487=1145.069,310.560,-74.989,-176.883,8.672,148.814
C02488=1145.073,310.312,-74.957,-176.886,8.668,148.813
C02489=1145.077,310.064,-74.926,-176.889,8.665,148.813
C02490=1145.081,309.816,-74.895,-176.891,8.661,148.813
C02491=1145.085,309.568,-74.863,-176.894,8.658,148.813
C02492=1145.090,309.321,-74.831,-176.897,8.654,148.813
C02493=1145.094,309.072,-74.800,-176.899,8.651,148.813
C02494=1145.098,308.825,-74.768,-176.902,8.648,148.813
C02495=1145.102,308.577,-74.736,-176.905,8.644,148.812
C02496=1145.106,308.328,-74.705,-176.907,8.640,148.812
C02497=1145.110,308.081,-74.674,-176.909,8.637,148.812
C02498=1145.114,307.833,-74.642,-176.913,8.633,148.812
C02499=1145.118,307.585,-74.611,-176.915,8.630,148.812
C02500=1145.123,307.336,-74.579,-176.917,8.627,148.812
C02501=1145.127,307.089,-74.547,-176.920,8.623,148.812
C02502=1145.131,306.840,-74.516,-176.923,8.620,148.812
C02503=1145.135,306.593,-74.484,-176.925,8.617,148.811
C02504=1145.139,306.344,-74.453,-176.928,8.613,148.811
C02505=1145.144,306.097,-74.422,-176.931,8.609,148.811
C02506=1145.147,305.849,-74.390,-176.933,8.606,148.811
C02507=1145.152,305.601,-74.359,-176.936,8.602,148.811
C02508=1145.156,305.353,-74.327,-176.939,8.599,148.811
C02509=1145.160,305.105,-74.297,-176.941,8.596,148.810
C02510=1145.164,304.857,-74.265,-176.944,8.592,148.810
C02511=1145.169,304.609,-74.234,-176.947,8.589,148.810
C02512=1145.173,304.360,-74.203,-176.949,8.585,148.810
C02513=1145.177,304.113,-74.171,-176.952,8.582,148.810
C02514=1145.181,303.864,-74.140,-176.955,8.578,148.810
C02515=1145.185,303.617,-74.109,-176.957,8.575,148.810
C02516=1145.189,303.368,-74.078,-176.959,8.572,148.810
C02517=1145.194,303.121,-74.046,-176.963,8.568,148.810
C02518=1145.198,302.872,-74.015,-176.965,8.565,148.809
C02519=1145.202,302.624,-73.984,-176.967,8.562,148.809
C02520=1145.207,302.377,-73.953,-176.971,8.558,148.809
C02521=1145.211,302.128,-73.922,-176.973,8.555,148.809
C02522=1145.214,301.881,-73.892,-176.975,8.551,148.809
C02523=1145.218,301.633,-73.860,-176.979,8.548,148.809
C02524=1145.223,301.385,-73.829,-176.981,8.544,148.809
C02525=1145.227,301.136,-73.798,-176.983,8.541,148.808
C02526=1145.231,300.888,-73.767,-176.987,8.537,148.808
C02527=1145.236,300.641,-73.736,-176.989,8.534,148.808
C02528=1145.240,300.392,-73.704,-176.991,8.531,148.808
C02529=1145.244,300.144,-73.674,-176.994,8.528,148.808
C02530=1145.248,299.896,-73.643,-176.997,8.524,148.808
C02531=1145.252,299.648,-73.612,-176.999,8.520,148.808
C02532=1145.257,299.400,-73.581,-177.002,8.517,148.808
C02533=1145.261,299.152,-73.550,-177.005,8.513,148.808
C02534=1145.264,298.904,-73.520,-177.008,8.510,148.808
C02535=1145.269,298.656,-73.489,-177.010,8.507,148.807
C02536=1145.273,298.408,-73.458,-177.012,8.504,148.807
C02537=1145.278,298.160,-73.427,-177.016,8.500,148.807
C02538=1145.282,297.912,-73.397,-177.018,8.497,148.807
C02539=1145.286,297.663,-73.366,-177.020,8.494,148.807
C02540=1145.290,297.415,-73.335,-177.023,8.491,148.807
C02541=1145.294,297.168,-73.303,-177.026,8.487,148.807
C02542=1145.298,296.920,-73.273,-177.029,8.484,148.807
C02543=1145.302,296.672,-73.242,-177.031,8.480,148.807
C02544=1145.307,296.424,-73.211,-177.034,8.476,148.806
C02545=1145.310,296.175,-73.181,-177.037,8.473,148.806
C02546=1145.315,295.927,-73.150,-177.039,8.470,148.806
C02547=1145.319,295.679,-73.119,-177.042,8.467,148.806
C02548=1145.324,295.431,-73.090,-177.045,8.463,148.806
C02549=1145.328,295.183,-73.059,-177.048,8.460,148.806
C02550=1145.332,294.935,-73.028,-177.050,8.457,148.806
C02551=1145.336,294.687,-72.998,-177.052,8.454,148.806
C02552=1145.340,294.438,-72.967,-177.056,8.450,148.806
C02553=1145.344,294.191,-72.936,-177.058,8.447,148.806
C02554=1145.349,293.943,-72.906,-177.061,8.444,148.806
C02555=1145.353,293.695,-72.875,-177.063,8.440,148.805
C02556=1145.357,293.446,-72.844,-177.067,8.437,148.805
C02557=1145.361,293.198,-72.814,-177.069,8.433,148.805
C02558=1145.365,292.950,-72.784,-177.072,8.430,148.805
C02559=1145.370,292.702,-72.753,-177.074,8.427,148.805
C02560=1145.373,292.454,-72.723,-177.077,8.423,148.805
C02561=1145.378,292.206,-72.692,-177.080,8.420,148.805
C02562=1145.382,291.958,-72.663,-177.082,8.417,148.805
C02563=1145.387,291.710,-72.632,-177.085,8.414,148.805
C02564=1145.390,291.462,-72.602,-177.088,8.410,148.805
C02565=1145.395,291.213,-72.571,-177.090,8.407,148.805
C02566=1145.399,290.965,-72.541,-177.093,8.404,148.804
C02567=1145.403,290.717,-72.510,-177.096,8.401,148.805
C02568=1145.407,290.469,-72.480,-177.098,8.398,148.804
C02569=1145.412,290.221,-72.450,-177.101,8.394,148.804
C02570=1145.415,289.973,-72.420,-177.104,8.390,148.804
C02571=1145.420,289.724,-72.390,-177.106,8.388,148.804
C02572=1145.424,289.476,-72.359,-177.109,8.384,148.804
C02573=1145.429,289.228,-72.329,-177.112,8.381,148.804
C02574=1145.433,288.980,-72.299,-177.114,8.377,148.804
C02575=1145.437,288.732,-72.269,-177.117,8.374,148.804
C02576=1145.442,288.484,-72.239,-177.120,8.371,148.804
C02577=1145.445,288.236,-72.208,-177.122,8.368,148.804
C02578=1145.450,287.987,-72.178,-177.125,8.364,148.804
C02579=1145.455,287.712,-72.145,-177.128,8.361,148.804
C02580=1145.459,287.437,-72.111,-177.131,8.357,148.804
C02581=1145.464,287.161,-72.079,-177.134,8.353,148.803
C02582=1145.469,286.886,-72.045,-177.137,8.350,148.803
C02583=1145.473,286.637,-72.015,-177.140,8.346,148.803
C02584=1145.476,286.390,-71.985,-177.143,8.343,148.803
C02585=1145.481,286.141,-71.955,-177.145,8.340,148.803
C02586=1145.485,285.893,-71.925,-177.148,8.337,148.803
C02587=1145.489,285.645,-71.895,-177.150,8.334,148.803
C02588=1145.494,285.397,-71.865,-177.153,8.331,148.803
C02589=1145.498,285.149,-71.835,-177.156,8.327,148.803
C02590=1145.502,284.901,-71.806,-177.159,8.324,148.803
C02591=1145.507,284.652,-71.776,-177.161,8.321,148.803
C02592=1145.511,284.404,-71.745,-177.164,8.318,148.803
C02593=1145.515,284.156,-71.716,-177.167,8.315,148.803
C02594=1145.520,283.908,-71.686,-177.169,8.311,148.803
C02595=1145.523,283.660,-71.656,-177.172,8.308,148.803
C02596=1145.528,283.412,-71.626,-177.175,8.305,148.803
C02597=1145.532,283.163,-71.597,-177.177,8.302,148.803
C02598=1145.537,282.915,-71.567,-177.180,8.299,148.803
C02599=1145.541,282.667,-71.537,-177.183,8.295,148.802
C02600=1145.545,282.419,-71.508,-177.186,8.292,148.802
C02601=1145.550,282.171,-71.478,-177.189,8.289,148.803
C02602=1145.554,281.922,-71.448,-177.191,8.285,148.802
C02603=1145.558,281.674,-71.419,-177.194,8.282,148.802
C02604=1145.562,281.426,-71.389,-177.196,8.279,148.802
C02605=1145.566,281.178,-71.359,-177.199,8.275,148.802
C02606=1145.570,280.930,-71.330,-177.202,8.273,148.802
C02607=1145.575,280.681,-71.300,-177.204,8.269,148.802
C02608=1145.579,280.433,-71.270,-177.207,8.266,148.802
C02609=1145.584,280.185,-71.241,-177.210,8.263,148.802
C02610=1145.588,279.937,-71.211,-177.212,8.260,148.802
C02611=1145.592,279.688,-71.182,-177.216,8.256,148.802
C02612=1145.596,279.440,-71.152,-177.218,8.253,148.802
C02613=1145.600,279.192,-71.123,-177.221,8.250,148.802
C02614=1145.604,278.943,-71.093,-177.224,8.247,148.802
C02615=1145.609,278.696,-71.064,-177.226,8.244,148.802
C02616=1145.613,278.448,-71.035,-177.229,8.241,148.802
C02617=1145.618,278.199,-71.005,-177.232,8.238,148.802
C02618=1145.622,277.951,-70.976,-177.234,8.234,148.802
C02619=1145.626,277.703,-70.947,-177.237,8.231,148.802
C02620=1145.630,277.455,-70.917,-177.240,8.228,148.802
C02621=1145.634,277.206,-70.888,-177.242,8.225,148.802
C02622=1145.638,276.958,-70.858,-177.245,8.222,148.802
C02623=1145.643,276.710,-70.829,-177.248,8.219,148.802
C02624=1145.647,276.461,-70.799,-177.250,8.216,148.802
C02625=1145.652,276.213,-70.771,-177.254,8.212,148.802
C02626=1145.656,275.965,-70.741,-177.256,8.209,148.802
C02627=1145.660,275.717,-70.712,-177.259,8.206,148.802
C02628=1145.664,275.468,-70.683,-177.261,8.203,148.802
C02629=1145.669,275.220,-70.653,-177.264,8.200,148.802
C02630=1145.673,274.972,-70.624,-177.267,8.197,148.801
C02631=1145.677,274.723,-70.595,-177.269,8.194,148.802
C02632=1145.682,274.476,-70.566,-177.272,8.191,148.802
C02633=1145.686,274.228,-70.537,-177.275,8.187,148.802
C02634=1145.690,273.979,-70.507,-177.278,8.184,148.801
C02635=1145.694,273.730,-70.479,-177.281,8.181,148.801
C02636=1145.698,273.482,-70.449,-177.283,8.178,148.802
C02637=1145.703,273.235,-70.420,-177.286,8.175,148.801
C02638=1145.708,272.986,-70.391,-177.288,8.172,148.801
C02639=1145.712,272.737,-70.362,-177.291,8.169,148.801
C02640=1145.715,272.489,-70.333,-177.294,8.166,148.802
C02641=1145.720,272.241,-70.304,-177.297,8.162,148.801
C02642=1145.725,271.993,-70.275,-177.300,8.159,148.801
C02643=1145.729,271.745,-70.246,-177.303,8.156,148.801
C02644=1145.733,271.496,-70.217,-177.305,8.153,148.802
C02645=1145.737,271.248,-70.188,-177.308,8.150,148.801
C02646=1145.742,271.000,-70.160,-177.310,8.147,148.801
C02647=1145.746,270.751,-70.130,-177.313,8.144,148.801
C02648=1145.750,270.503,-70.102,-177.316,8.141,148.801
C02649=1145.754,270.255,-70.073,-177.318,8.138,148.801
C02650=1145.759,270.007,-70.044,-177.321,8.135,148.801
C02651=1145.763,269.758,-70.015,-177.324,8.131,148.801
C02652=1145.767,269.510,-69.986,-177.327,8.128,148.802
C02653=1145.772,269.262,-69.958,-177.330,8.125,148.801
C02654=1145.776,269.013,-69.929,-177.332,8.122,148.801
C02655=1145.780,268.765,-69.900,-177.335,8.119,148.801
C02656=1145.785,268.517,-69.872,-177.338,8.116,148.802
C02657=1145.789,268.269,-69.842,-177.340,8.113,148.801
C02658=1145.793,268.020,-69.814,-177.343,8.110,148.801
C02659=1145.797,267.772,-69.785,-177.346,8.107,148.801
C02660=1145.802,267.524,-69.756,-177.349,8.104,148.802
C02661=1145.806,267.275,-69.728,-177.351,8.101,148.801
C02662=1145.810,267.027,-69.699,-177.354,8.097,148.801
C02663=1145.815,266.779,-69.670,-177.357,8.094,148.801
C02664=1145.819,266.530,-69.642,-177.360,8.091,148.802
C02665=1145.823,266.283,-69.613,-177.363,8.088,148.802
C02666=1145.828,266.034,-69.584,-177.365,8.085,148.801
C02667=1145.832,265.785,-69.556,-177.368,8.082,148.801
C02668=1145.837,265.537,-69.528,-177.371,8.079,148.802
C02669=1145.841,265.289,-69.498,-177.373,8.076,148.802
C02670=1145.845,265.040,-69.470,-177.376,8.073,148.802
C02671=1145.850,264.792,-69.442,-177.379,8.070,148.802
C02672=1145.854,264.543,-69.414,-177.381,8.067,148.802
C02673=1145.858,264.296,-69.385,-177.384,8.064,148.802
C02674=1145.862,264.047,-69.357,-177.387,8.061,148.802
C02675=1145.867,263.798,-69.328,-177.390,8.058,148.802
C02676=1145.871,263.550,-69.300,-177.392,8.055,148.802
C02677=1145.875,263.301,-69.271,-177.395,8.052,148.802
C02678=1145.880,263.054,-69.244,-177.398,8.048,148.802
C02679=1145.884,262.805,-69.215,-177.401,8.045,148.802
C02680=1145.888,262.557,-69.186,-177.404,8.042,148.802
C02681=1145.893,262.309,-69.158,-177.406,8.039,148.802
C02682=1145.897,262.061,-69.130,-177.409,8.037,148.802
C02683=1145.902,261.786,-69.098,-177.412,8.034,148.802
C02684=1145.907,261.513,-69.068,-177.415,8.030,148.802
C02685=1145.911,261.240,-69.037,-177.418,8.027,148.802
C02686=1145.916,260.967,-69.005,-177.421,8.023,148.802
C02687=1145.920,260.718,-68.977,-177.424,8.020,148.802
C02688=1145.925,260.470,-68.948,-177.427,8.017,148.802
C02689=1145.929,260.221,-68.920,-177.429,8.014,148.802
C02690=1145.934,259.973,-68.893,-177.432,8.011,148.802
C02691=1145.938,259.724,-68.864,-177.435,8.008,148.802
C02692=1145.942,259.476,-68.837,-177.438,8.005,148.802
C02693=1145.946,259.227,-68.808,-177.441,8.002,148.802
C02694=1145.951,258.979,-68.780,-177.443,7.999,148.802
C02695=1145.955,258.731,-68.752,-177.446,7.996,148.802
C02696=1145.959,258.483,-68.724,-177.448,7.993,148.802
C02697=1145.964,258.234,-68.695,-177.451,7.990,148.802
C02698=1145.968,257.986,-68.668,-177.454,7.987,148.802
C02699=1145.972,257.737,-68.640,-177.457,7.984,148.803
C02700=1145.977,257.489,-68.612,-177.460,7.981,148.803
C02701=1145.982,257.241,-68.584,-177.462,7.979,148.803
C02702=1145.985,256.992,-68.556,-177.465,7.976,148.803
C02703=1145.990,256.744,-68.528,-177.467,7.972,148.803
C02704=1145.995,256.495,-68.500,-177.470,7.969,148.803
C02705=1145.999,256.247,-68.472,-177.473,7.967,148.803
C02706=1146.003,255.998,-68.444,-177.476,7.964,148.803
C02707=1146.007,255.750,-68.416,-177.479,7.961,148.803
C02708=1146.012,255.502,-68.389,-177.481,7.958,148.803
C02709=1146.016,255.253,-68.361,-177.484,7.955,148.803
C02710=1146.021,255.005,-68.333,-177.487,7.952,148.803
C02711=1146.025,254.756,-68.305,-177.490,7.949,148.803
C02712=1146.029,254.508,-68.278,-177.493,7.946,148.803
C02713=1146.034,254.260,-68.249,-177.495,7.943,148.803
C02714=1146.038,254.011,-68.222,-177.498,7.940,148.803
C02715=1146.042,253.763,-68.194,-177.501,7.937,148.803
C02716=1146.047,253.515,-68.166,-177.503,7.934,148.803
C02717=1146.051,253.266,-68.139,-177.506,7.931,148.803
C02718=1146.055,253.018,-68.111,-177.509,7.928,148.803
C02719=1146.059,252.769,-68.084,-177.512,7.925,148.803
C02720=1146.064,252.521,-68.055,-177.514,7.922,148.803
C02721=1146.069,252.272,-68.028,-177.517,7.919,148.804
C02722=1146.073,252.023,-68.000,-177.520,7.916,148.804
C02723=1146.077,251.776,-67.972,-177.523,7.913,148.804
C02724=1146.082,251.527,-67.945,-177.526,7.911,148.804
C02725=1146.086,251.278,-67.918,-177.528,7.908,148.804
C02726=1146.090,251.030,-67.890,-177.531,7.905,148.804
C02727=1146.095,250.782,-67.863,-177.534,7.902,148.804
C02728=1146.099,250.534,-67.835,-177.537,7.899,148.804
C02729=1146.103,250.284,-67.808,-177.539,7.896,148.804
C02730=1146.108,250.037,-67.780,-177.542,7.893,148.804
C02731=1146.112,249.788,-67.753,-177.545,7.890,148.804
C02732=1146.116,249.539,-67.726,-177.548,7.887,148.804
C02733=1146.121,249.291,-67.698,-177.551,7.884,148.804
C02734=1146.125,249.043,-67.671,-177.553,7.881,148.804
C02735=1146.130,248.795,-67.643,-177.556,7.879,148.805
C02736=1146.134,248.545,-67.615,-177.558,7.876,148.805
C02737=1146.138,248.297,-67.588,-177.561,7.873,148.805
C02738=1146.143,248.049,-67.561,-177.564,7.870,148.805
C02739=1146.147,247.801,-67.534,-177.567,7.867,148.805
C02740=1146.151,247.551,-67.506,-177.570,7.865,148.805
C02741=1146.156,247.303,-67.479,-177.572,7.862,148.805
C02742=1146.160,247.055,-67.451,-177.575,7.859,148.805
C02743=1146.165,246.807,-67.424,-177.578,7.856,148.805
C02744=1146.170,246.558,-67.397,-177.581,7.853,148.805
C02745=1146.174,246.309,-67.370,-177.583,7.850,148.805
C02746=1146.177,246.061,-67.343,-177.586,7.847,148.805
C02747=1146.182,245.813,-67.316,-177.589,7.844,148.805
C02748=1146.187,245.564,-67.288,-177.592,7.841,148.806
C02749=1146.191,245.316,-67.261,-177.595,7.838,148.806
C02750=1146.195,245.067,-67.234,-177.597,7.835,148.806
C02751=1146.200,244.818,-67.207,-177.600,7.832,148.806
C02752=1146.205,244.570,-67.180,-177.603,7.829,148.806
C02753=1146.208,244.322,-67.153,-177.605,7.827,148.806
C02754=1146.213,244.074,-67.126,-177.608,7.824,148.806
C02755=1146.218,243.825,-67.099,-177.611,7.821,148.806
C02756=1146.222,243.576,-67.071,-177.614,7.819,148.806
C02757=1146.226,243.327,-67.044,-177.616,7.816,148.806
C02758=1146.230,243.079,-67.018,-177.619,7.813,148.806
C02759=1146.235,242.831,-66.991,-177.622,7.810,148.806
C02760=1146.240,242.582,-66.963,-177.625,7.807,148.806
C02761=1146.244,242.334,-66.936,-177.628,7.804,148.807
C02762=1146.248,242.086,-66.910,-177.630,7.801,148.807
C02763=1146.252,241.836,-66.883,-177.633,7.798,148.807
C02764=1146.257,241.588,-66.855,-177.636,7.795,148.807
C02765=1146.262,241.339,-66.828,-177.639,7.793,148.807
C02766=1146.266,241.091,-66.802,-177.641,7.790,148.807
C02767=1146.270,240.843,-66.775,-177.644,7.788,148.807
C02768=1146.275,240.594,-66.748,-177.647,7.785,148.807
C02769=1146.279,240.345,-66.722,-177.650,7.782,148.807
C02770=1146.284,240.097,-66.695,-177.653,7.779,148.807
C02771=1146.288,239.848,-66.668,-177.655,7.776,148.808
C02772=1146.292,239.600,-66.641,-177.658,7.773,148.808
C02773=1146.297,239.352,-66.614,-177.661,7.770,148.808
C02774=1146.302,239.103,-66.587,-177.664,7.767,148.808
C02775=1146.306,238.855,-66.561,-177.666,7.765,148.808
C02776=1146.310,238.606,-66.535,-177.669,7.762,148.808
C02777=1146.315,238.357,-66.507,-177.671,7.759,148.808
C02778=1146.319,238.109,-66.481,-177.675,7.757,148.808
C02779=1146.323,237.860,-66.454,-177.677,7.754,148.808
C02780=1146.327,237.611,-66.428,-177.680,7.751,148.808
C02781=1146.332,237.363,-66.401,-177.683,7.748,148.809
C02782=1146.337,237.114,-66.374,-177.686,7.745,148.809
C02783=1146.341,236.866,-66.347,-177.689,7.742,148.809
C02784=1146.346,236.617,-66.321,-177.691,7.740,148.809
C02785=1146.349,236.369,-66.294,-177.694,7.737,148.809
C02786=1146.354,236.120,-66.267,-177.696,7.734,148.809
C02787=1146.359,235.848,-66.239,-177.700,7.731,148.809
C02788=1146.364,235.577,-66.210,-177.703,7.728,148.809
C02789=1146.369,235.305,-66.181,-177.706,7.725,148.809
C02790=1146.374,235.033,-66.153,-177.709,7.722,148.810
C02791=1146.378,234.785,-66.126,-177.711,7.719,148.810
C02792=1146.383,234.536,-66.100,-177.715,7.716,148.810
C02793=1146.387,234.287,-66.073,-177.717,7.713,148.810
C02794=1146.391,234.039,-66.046,-177.720,7.710,148.810
C02795=1146.396,233.790,-66.020,-177.722,7.708,148.810
C02796=1146.400,233.542,-65.993,-177.725,7.705,148.810
C02797=1146.405,233.293,-65.967,-177.728,7.703,148.810
C02798=1146.409,233.045,-65.941,-177.731,7.700,148.810
C02799=1146.413,232.796,-65.915,-177.734,7.697,148.811
C02800=1146.418,232.547,-65.888,-177.737,7.694,148.811
C02801=1146.422,232.299,-65.862,-177.740,7.691,148.811
C02802=1146.427,232.049,-65.836,-177.742,7.689,148.811
C02803=1146.432,231.802,-65.810,-177.745,7.686,148.811
C02804=1146.436,231.553,-65.784,-177.748,7.683,148.811
C02805=1146.440,231.305,-65.757,-177.750,7.680,148.811
C02806=1146.445,231.056,-65.731,-177.754,7.678,148.812
C02807=1146.449,230.807,-65.704,-177.756,7.675,148.812
C02808=1146.454,230.559,-65.678,-177.759,7.673,148.812
C02809=1146.458,230.310,-65.652,-177.761,7.670,148.812
C02810=1146.463,230.062,-65.626,-177.764,7.667,148.812
C02811=1146.467,229.813,-65.600,-177.767,7.664,148.812
C02812=1146.471,229.564,-65.574,-177.770,7.661,148.812
C02813=1146.475,229.316,-65.548,-177.773,7.658,148.812
C02814=1146.480,229.067,-65.521,-177.775,7.656,148.813
C02815=1146.485,228.818,-65.496,-177.778,7.653,148.813
C02816=1146.489,228.570,-65.470,-177.781,7.651,148.813
C02817=1146.494,228.322,-65.443,-177.784,7.648,148.813
C02818=1146.498,228.073,-65.418,-177.787,7.645,148.813
C02819=1146.502,227.824,-65.392,-177.789,7.643,148.813
C02820=1146.507,227.575,-65.366,-177.792,7.640,148.813
C02821=1146.512,227.326,-65.340,-177.795,7.637,148.813
C02822=1146.516,227.079,-65.314,-177.797,7.634,148.813
C02823=1146.520,226.830,-65.288,-177.801,7.632,148.814
C02824=1146.525,226.581,-65.262,-177.803,7.629,148.814
C02825=1146.529,226.332,-65.236,-177.806,7.627,148.814
C02826=1146.534,226.084,-65.210,-177.808,7.624,148.814
C02827=1146.539,225.835,-65.185,-177.811,7.621,148.814
C02828=1146.543,225.586,-65.159,-177.815,7.618,148.814
C02829=1146.547,225.338,-65.132,-177.817,7.616,148.815
C02830=1146.552,225.090,-65.107,-177.820,7.613,148.815
C02831=1146.556,224.841,-65.081,-177.822,7.610,148.815
C02832=1146.561,224.592,-65.055,-177.825,7.607,148.815
C02833=1146.565,224.343,-65.029,-177.828,7.605,148.815
C02834=1146.570,224.095,-65.004,-177.831,7.603,148.815
C02835=1146.574,223.846,-64.978,-177.833,7.600,148.815
C02836=1146.578,223.597,-64.952,-177.836,7.597,148.815
C02837=1146.583,223.349,-64.926,-177.839,7.594,148.816
C02838=1146.587,223.101,-64.901,-177.842,7.591,148.816
C02839=1146.592,222.852,-64.875,-177.844,7.589,148.816
C02840=1146.596,222.603,-64.850,-177.847,7.586,148.816
C02841=1146.601,222.355,-64.824,-177.850,7.584,148.816
C02842=1146.605,222.106,-64.798,-177.853,7.581,148.816
C02843=1146.610,221.857,-64.772,-177.855,7.579,148.817
C02844=1146.615,221.608,-64.747,-177.858,7.576,148.817
C02845=1146.619,221.359,-64.722,-177.862,7.573,148.817
C02846=1146.623,221.111,-64.696,-177.864,7.570,148.817
C02847=1146.628,220.862,-64.671,-177.867,7.568,148.817
C02848=1146.632,220.614,-64.645,-177.869,7.565,148.817
C02849=1146.637,220.365,-64.619,-177.873,7.563,148.818
C02850=1146.642,220.117,-64.594,-177.875,7.560,148.818
C02851=1146.646,219.867,-64.569,-177.878,7.558,148.818
C02852=1146.650,219.619,-64.543,-177.880,7.555,148.818
C02853=1146.654,219.371,-64.518,-177.884,7.552,148.818
C02854=1146.659,219.122,-64.492,-177.886,7.549,148.818
C02855=1146.664,218.873,-64.468,-177.889,7.547,148.818
C02856=1146.668,218.624,-64.442,-177.891,7.544,148.819
C02857=1146.672,218.376,-64.416,-177.895,7.542,148.819
C02858=1146.677,218.127,-64.391,-177.898,7.539,148.819
C02859=1146.682,217.878,-64.366,-177.900,7.537,148.819
C02860=1146.686,217.630,-64.340,-177.903,7.534,148.819
C02861=1146.691,217.381,-64.315,-177.906,7.531,148.819
C02862=1146.695,217.132,-64.290,-177.909,7.528,148.820
C02863=1146.699,216.884,-64.265,-177.911,7.526,148.820
C02864=1146.703,216.635,-64.239,-177.914,7.524,148.820
C02865=1146.709,216.386,-64.214,-177.917,7.521,148.820
C02866=1146.713,216.138,-64.189,-177.919,7.519,148.820
C02867=1146.718,215.890,-64.163,-177.922,7.516,148.821
C02868=1146.722,215.640,-64.138,-177.925,7.513,148.821
C02869=1146.727,215.392,-64.113,-177.928,7.510,148.821
C02870=1146.731,215.143,-64.088,-177.931,7.508,148.821
C02871=1146.735,214.894,-64.063,-177.933,7.505,148.821
C02872=1146.740,214.645,-64.038,-177.936,7.503,148.821
C02873=1146.744,214.397,-64.012,-177.938,7.500,148.821
C02874=1146.749,214.148,-63.988,-177.942,7.498,148.822
C02875=1146.753,213.899,-63.962,-177.944,7.495,148.822
C02876=1146.758,213.651,-63.938,-177.947,7.492,148.822
C02877=1146.762,213.402,-63.912,-177.950,7.490,148.822
C02878=1146.767,213.153,-63.888,-177.953,7.487,148.822
C02879=1146.771,212.905,-63.862,-177.956,7.484,148.822
C02880=1146.776,212.656,-63.837,-177.958,7.483,148.823
C02881=1146.780,212.407,-63.812,-177.961,7.480,148.823
C02882=1146.785,212.159,-63.788,-177.964,7.477,148.823
C02883=1146.790,211.910,-63.763,-177.967,7.475,148.823
C02884=1146.794,211.661,-63.737,-177.969,7.472,148.823
C02885=1146.798,211.413,-63.713,-177.973,7.470,148.824
C02886=1146.803,211.163,-63.688,-177.975,7.468,148.824
C02887=1146.808,210.915,-63.663,-177.978,7.465,148.824
C02888=1146.812,210.666,-63.638,-177.981,7.462,148.824
C02889=1146.817,210.417,-63.614,-177.983,7.460,148.824
C02890=1146.821,210.169,-63.588,-177.986,7.457,148.824
C02891=1146.826,209.898,-63.561,-177.989,7.455,148.825
C02892=1146.831,209.627,-63.534,-177.992,7.452,148.825
C02893=1146.836,209.357,-63.507,-177.995,7.449,148.825
C02894=1146.840,209.086,-63.480,-177.998,7.446,148.825
C02895=1146.845,208.838,-63.456,-178.001,7.444,148.826
C02896=1146.850,208.589,-63.432,-178.003,7.441,148.826
C02897=1146.854,208.340,-63.407,-178.006,7.439,148.826
C02898=1146.859,208.092,-63.381,-178.010,7.436,148.826
C02899=1146.863,207.843,-63.357,-178.012,7.434,148.826
C02900=1146.868,207.594,-63.332,-178.015,7.431,148.827
C02901=1146.873,207.346,-63.308,-178.018,7.428,148.827
C02902=1146.877,207.096,-63.283,-178.020,7.426,148.827
C02903=1146.881,206.848,-63.259,-178.023,7.424,148.827
C02904=1146.887,206.599,-63.234,-178.026,7.421,148.827
C02905=1146.890,206.350,-63.209,-178.028,7.419,148.827
C02906=1146.895,206.102,-63.184,-178.032,7.416,148.828
C02907=1146.900,205.853,-63.160,-178.034,7.413,148.828
C02908=1146.904,205.604,-63.135,-178.037,7.411,148.828
C02909=1146.909,205.355,-63.111,-178.040,7.409,148.828
C02910=1146.914,205.107,-63.086,-178.043,7.407,148.829
C02911=1146.917,204.858,-63.062,-178.045,7.404,148.829
C02912=1146.923,204.609,-63.037,-178.048,7.401,148.829
C02913=1146.927,204.361,-63.013,-178.051,7.399,148.829
C02914=1146.932,204.111,-62.988,-178.054,7.396,148.829
C02915=1146.936,203.863,-62.964,-178.057,7.394,148.830
C02916=1146.941,203.614,-62.940,-178.059,7.392,148.830
C02917=1146.945,203.366,-62.915,-178.062,7.389,148.830
C02918=1146.949,203.116,-62.891,-178.065,7.386,148.830
C02919=1146.954,202.868,-62.866,-178.067,7.384,148.830
C02920=1146.959,202.619,-62.842,-178.071,7.382,148.831
C02921=1146.963,202.370,-62.817,-178.073,7.379,148.831
C02922=1146.968,202.121,-62.794,-178.076,7.377,148.831
C02923=1146.972,201.872,-62.770,-178.079,7.374,148.831
C02924=1146.978,201.624,-62.745,-178.082,7.372,148.832
C02925=1146.981,201.375,-62.721,-178.084,7.369,148.832
C02926=1146.986,201.126,-62.697,-178.087,7.367,148.832
C02927=1146.991,200.877,-62.672,-178.090,7.365,148.832
C02928=1146.995,200.629,-62.648,-178.093,7.362,148.832
C02929=1147.000,200.380,-62.625,-178.095,7.360,148.833
C02930=1147.004,200.131,-62.599,-178.098,7.357,148.833
C02931=1147.009,199.882,-62.575,-178.101,7.355,148.833
C02932=1147.013,199.634,-62.551,-178.104,7.352,148.833
C02933=1147.018,199.385,-62.528,-178.107,7.350,148.833
C02934=1147.022,199.135,-62.503,-178.109,7.348,148.834
C02935=1147.027,198.887,-62.479,-178.112,7.345,148.834
C02936=1147.031,198.638,-62.455,-178.115,7.343,148.834
C02937=1147.036,198.389,-62.431,-178.118,7.341,148.834
C02938=1147.041,198.141,-62.407,-178.120,7.338,148.835
C02939=1147.045,197.892,-62.383,-178.123,7.336,148.835
C02940=1147.050,197.643,-62.359,-178.126,7.333,148.835
C02941=1147.054,197.394,-62.335,-178.128,7.331,148.835
C02942=1147.058,197.146,-62.311,-178.132,7.328,148.835
C02943=1147.064,196.896,-62.287,-178.134,7.326,148.836
C02944=1147.068,196.648,-62.263,-178.137,7.324,148.836
C02945=1147.073,196.400,-62.239,-178.139,7.322,148.836
C02946=1147.077,196.151,-62.215,-178.143,7.319,148.836
C02947=1147.081,195.901,-62.191,-178.146,7.316,148.836
C02948=1147.087,195.652,-62.167,-178.148,7.314,148.837
C02949=1147.091,195.404,-62.143,-178.151,7.311,148.837
C02950=1147.096,195.155,-62.120,-178.154,7.310,148.837
C02951=1147.100,194.906,-62.095,-178.157,7.307,148.837
C02952=1147.105,194.657,-62.072,-178.159,7.305,148.838
C02953=1147.109,194.409,-62.048,-178.162,7.302,148.838
C02954=1147.114,194.160,-62.025,-178.165,7.300,148.838
C02955=1147.118,193.911,-62.001,-178.168,7.298,148.839
C02956=1147.123,193.662,-61.977,-178.171,7.295,148.839
C02957=1147.127,193.413,-61.952,-178.173,7.293,148.839
C02958=1147.132,193.164,-61.929,-178.176,7.290,148.839
C02959=1147.137,192.915,-61.905,-178.179,7.289,148.839
C02960=1147.141,192.666,-61.881,-178.182,7.286,148.840
C02961=1147.146,192.417,-61.858,-178.184,7.284,148.840
C02962=1147.150,192.169,-61.834,-178.187,7.281,148.840
C02963=1147.155,191.920,-61.811,-178.190,7.279,148.840
C02964=1147.159,191.672,-61.787,-178.193,7.276,148.841
C02965=1147.164,191.422,-61.763,-178.195,7.275,148.841
C02966=1147.169,191.173,-61.740,-178.198,7.272,148.841
C02967=1147.173,190.925,-61.716,-178.201,7.270,148.841
C02968=1147.178,190.676,-61.692,-178.204,7.267,148.841
C02969=1147.183,190.427,-61.669,-178.206,7.265,148.842
C02970=1147.187,190.179,-61.645,-178.210,7.263,148.842
C02971=1147.192,189.930,-61.622,-178.213,7.260,148.842
C02972=1147.196,189.680,-61.598,-178.215,7.258,148.843
C02973=1147.201,189.431,-61.575,-178.218,7.255,148.843
C02974=1147.206,189.183,-61.551,-178.221,7.253,148.843
C02975=1147.210,188.934,-61.527,-178.224,7.251,148.843
C02976=1147.215,188.685,-61.504,-178.226,7.249,148.844
C02977=1147.220,188.436,-61.481,-178.229,7.246,148.844
C02978=1147.224,188.187,-61.458,-178.232,7.244,148.844
C02979=1147.228,187.939,-61.434,-178.235,7.242,148.844
C02980=1147.233,187.690,-61.411,-178.237,7.240,148.845
C02981=1147.237,187.441,-61.387,-178.240,7.237,148.845
C02982=1147.242,187.192,-61.364,-178.243,7.235,148.845
C02983=1147.247,186.943,-61.341,-178.246,7.232,148.845
C02984=1147.252,186.694,-61.317,-178.249,7.231,148.846
C02985=1147.257,186.445,-61.294,-178.251,7.228,148.846
C02986=1147.261,186.197,-61.271,-178.254,7.226,148.846
C02987=1147.265,185.948,-61.247,-178.256,7.224,148.846
C02988=1147.270,185.699,-61.224,-178.260,7.221,148.847
C02989=1147.275,185.450,-61.201,-178.262,7.220,148.847
C02990=1147.279,185.201,-61.177,-178.265,7.217,148.847
C02991=1147.283,184.952,-61.154,-178.268,7.215,148.847
C02992=1147.288,184.703,-61.131,-178.271,7.212,148.848
C02993=1147.293,184.454,-61.108,-178.273,7.210,148.848
C02994=1147.298,184.206,-61.085,-178.277,7.208,148.848
C02995=1147.303,183.935,-61.059,-178.279,7.205,148.848
C02996=1147.307,183.666,-61.035,-178.282,7.203,148.849
C02997=1147.312,183.396,-61.010,-178.285,7.201,148.849
C02998=1147.318,183.127,-60.984,-178.289,7.198,148.849
C02999=1147.321,182.878,-60.961,-178.291,7.196,148.850
C03000=1147.326,182.629,-60.939,-178.294,7.193,148.850
C03001=1147.332,182.380,-60.916,-178.296,7.191,148.850
C03002=1147.336,182.131,-60.892,-178.300,7.189,148.850
C03003=1147.340,181.883,-60.870,-178.302,7.187,148.851
C03004=1147.345,181.634,-60.846,-178.305,7.184,148.851
C03005=1147.350,181.385,-60.823,-178.308,7.182,148.851
C03006=1147.354,181.136,-60.800,-178.311,7.181,148.852
C03007=1147.359,180.888,-60.777,-178.313,7.178,148.852
C03008=1147.364,180.638,-60.754,-178.316,7.176,148.852
C03009=1147.368,180.389,-60.732,-178.319,7.173,148.852
C03010=1147.373,180.140,-60.708,-178.322,7.171,148.853
C03011=1147.377,179.891,-60.685,-178.325,7.169,148.853
C03012=1147.382,179.643,-60.663,-178.327,7.167,148.853
C03013=1147.387,179.393,-60.640,-178.330,7.164,148.853
C03014=1147.391,179.145,-60.617,-178.333,7.162,148.854
C03015=1147.396,178.896,-60.594,-178.335,7.160,148.854
C03016=1147.401,178.646,-60.571,-178.339,7.158,148.854
C03017=1147.405,178.398,-60.549,-178.341,7.156,148.855
C03018=1147.410,178.149,-60.525,-178.344,7.153,148.855
C03019=1147.414,177.900,-60.503,-178.347,7.151,148.855
C03020=1147.419,177.651,-60.480,-178.350,7.149,148.856
C03021=1147.424,177.403,-60.458,-178.352,7.147,148.856
C03022=1147.428,177.154,-60.434,-178.355,7.145,148.856
C03023=1147.432,176.904,-60.412,-178.358,7.142,148.856
C03024=1147.438,176.656,-60.389,-178.360,7.140,148.857
C03025=1147.442,176.407,-60.367,-178.364,7.138,148.857
C03026=1147.447,176.158,-60.344,-178.366,7.136,148.857
C03027=1147.451,175.909,-60.321,-178.369,7.134,148.857
C03028=1147.456,175.660,-60.299,-178.372,7.131,148.858
C03029=1147.460,175.411,-60.276,-178.375,7.130,148.858
C03030=1147.465,175.161,-60.253,-178.377,7.127,148.858
C03031=1147.470,174.913,-60.231,-178.380,7.125,148.859
C03032=1147.475,174.664,-60.208,-178.383,7.123,148.859
C03033=1147.479,174.415,-60.186,-178.386,7.121,148.859
C03034=1147.484,174.166,-60.163,-178.388,7.119,148.859
C03035=1147.488,173.917,-60.140,-178.392,7.116,148.860
C03036=1147.493,173.668,-60.118,-178.394,7.114,148.860
C03037=1147.498,173.420,-60.095,-178.397,7.112,148.860
C03038=1147.502,173.170,-60.073,-178.400,7.110,148.861
C03039=1147.507,172.921,-60.050,-178.403,7.108,148.861
C03040=1147.512,172.673,-60.028,-178.405,7.105,148.861
C03041=1147.516,172.424,-60.005,-178.408,7.103,148.862
C03042=1147.521,172.174,-59.983,-178.411,7.102,148.862
C03043=1147.526,171.926,-59.961,-178.414,7.099,148.862
C03044=1147.530,171.677,-59.938,-178.416,7.097,148.862
C03045=1147.535,171.428,-59.916,-178.419,7.095,148.863
C03046=1147.540,171.178,-59.894,-178.422,7.093,148.863
C03047=1147.544,170.930,-59.871,-178.424,7.091,148.863
C03048=1147.549,170.681,-59.849,-178.427,7.089,148.864
C03049=1147.554,170.431,-59.826,-178.430,7.086,148.864
C03050=1147.559,170.183,-59.804,-178.433,7.085,148.864
C03051=1147.563,169.934,-59.782,-178.436,7.082,148.864
C03052=1147.567,169.685,-59.760,-178.439,7.080,148.865
C03053=1147.572,169.436,-59.737,-178.441,7.078,148.865
C03054=1147.577,169.187,-59.715,-178.445,7.076,148.866
C03055=1147.582,168.938,-59.693,-178.447,7.074,148.866
C03056=1147.587,168.689,-59.671,-178.450,7.072,148.866
C03057=1147.591,168.441,-59.648,-178.453,7.069,148.866
C03058=1147.595,168.191,-59.626,-178.456,7.068,148.867
C03059=1147.600,167.942,-59.604,-178.458,7.066,148.867
C03060=1147.605,167.693,-59.582,-178.461,7.063,148.867
C03061=1147.610,167.444,-59.560,-178.464,7.061,148.868
C03062=1147.614,167.196,-59.537,-178.466,7.060,148.868
C03063=1147.618,166.946,-59.515,-178.469,7.057,148.868
C03064=1147.624,166.697,-59.493,-178.472,7.055,148.869
C03065=1147.628,166.448,-59.471,-178.475,7.053,148.869
C03066=1147.633,166.199,-59.449,-178.478,7.051,148.869
C03067=1147.637,165.950,-59.427,-178.480,7.049,148.869
C03068=1147.642,165.701,-59.406,-178.483,7.047,148.870
C03069=1147.647,165.452,-59.384,-178.486,7.044,148.870
C03070=1147.652,165.203,-59.361,-178.489,7.043,148.871
C03071=1147.656,164.954,-59.339,-178.491,7.041,148.871
C03072=1147.661,164.706,-59.317,-178.494,7.038,148.871
C03073=1147.665,164.456,-59.295,-178.497,7.036,148.871
C03074=1147.670,164.208,-59.273,-178.500,7.035,148.872
C03075=1147.674,163.958,-59.251,-178.503,7.032,148.872
C03076=1147.679,163.710,-59.229,-178.505,7.030,148.872
C03077=1147.684,163.461,-59.208,-178.508,7.028,148.873
C03078=1147.688,163.212,-59.186,-178.511,7.026,148.873
C03079=1147.694,162.963,-59.163,-178.514,7.024,148.873
C03080=1147.698,162.714,-59.141,-178.517,7.022,148.874
C03081=1147.703,162.464,-59.120,-178.519,7.020,148.874
C03082=1147.708,162.215,-59.098,-178.522,7.018,148.874
C03083=1147.713,161.966,-59.077,-178.525,7.016,148.875
C03084=1147.717,161.718,-59.055,-178.528,7.014,148.875
C03085=1147.722,161.468,-59.033,-178.531,7.012,148.875
C03086=1147.727,161.220,-59.011,-178.533,7.010,148.876
C03087=1147.731,160.970,-58.989,-178.536,7.008,148.876
C03088=1147.736,160.722,-58.967,-178.539,7.005,148.876
C03089=1147.740,160.472,-58.945,-178.542,7.004,148.877
C03090=1147.745,160.223,-58.924,-178.545,7.002,148.877
C03091=1147.750,159.974,-58.903,-178.547,7.000,148.877
C03092=1147.754,159.725,-58.881,-178.550,6.997,148.878
C03093=1147.759,159.476,-58.859,-178.553,6.996,148.878
C03094=1147.764,159.228,-58.837,-178.555,6.994,148.878
C03095=1147.769,158.978,-58.816,-178.558,6.992,148.879
C03096=1147.773,158.729,-58.794,-178.561,6.989,148.879
C03097=1147.778,158.481,-58.773,-178.564,6.987,148.879
C03098=1147.783,158.231,-58.751,-178.566,6.986,148.880
C03099=1147.787,157.962,-58.728,-178.570,6.983,148.880
C03100=1147.793,157.693,-58.705,-178.572,6.981,148.880
C03101=1147.797,157.424,-58.681,-178.576,6.979,148.881
C03102=1147.803,157.155,-58.658,-178.578,6.977,148.881
C03103=1147.808,156.906,-58.636,-178.582,6.975,148.881
C03104=1147.812,156.657,-58.616,-178.584,6.973,148.882
C03105=1147.816,156.408,-58.594,-178.587,6.971,148.882
C03106=1147.821,156.159,-58.572,-178.589,6.969,148.882
C03107=1147.826,155.910,-58.551,-178.593,6.967,148.883
C03108=1147.831,155.662,-58.529,-178.595,6.965,148.883
C03109=1147.836,155.412,-58.508,-178.598,6.963,148.883
C03110=1147.841,155.163,-58.486,-178.601,6.961,148.884
C03111=1147.845,154.915,-58.465,-178.604,6.959,148.884
C03112=1147.849,154.665,-58.444,-178.606,6.957,148.884
C03113=1147.854,154.416,-58.422,-178.609,6.955,148.885
C03114=1147.859,154.167,-58.401,-178.612,6.953,148.885
C03115=1147.864,153.918,-58.379,-178.615,6.951,148.885
C03116=1147.868,153.668,-58.359,-178.618,6.949,148.886
C03117=1147.873,153.420,-58.337,-178.620,6.947,148.886
C03118=1147.878,153.171,-58.316,-178.623,6.946,148.887
C03119=1147.883,152.922,-58.294,-178.626,6.943,148.887
C03120=1147.888,152.673,-58.273,-178.629,6.941,148.887
C03121=1147.892,152.424,-58.252,-178.631,6.939,148.888
C03122=1147.897,152.174,-58.231,-178.634,6.938,148.888
C03123=1147.902,151.926,-58.209,-178.637,6.936,148.888
C03124=1147.907,151.677,-58.188,-178.640,6.933,148.889
C03125=1147.911,151.427,-58.168,-178.643,6.932,148.889
C03126=1147.916,151.178,-58.146,-178.645,6.930,148.889
C03127=1147.921,150.929,-58.125,-178.648,6.928,148.890
C03128=1147.925,150.681,-58.104,-178.650,6.926,148.890
C03129=1147.930,150.431,-58.083,-178.654,6.924,148.890
C03130=1147.935,150.182,-58.062,-178.656,6.922,148.891
C03131=1147.939,149.933,-58.041,-178.659,6.920,148.891
C03132=1147.944,149.684,-58.020,-178.662,6.918,148.891
C03133=1147.949,149.435,-57.999,-178.665,6.916,148.892
C03134=1147.953,149.186,-57.977,-178.668,6.914,148.892
C03135=1147.959,148.937,-57.957,-178.671,6.912,148.893
C03136=1147.964,148.688,-57.936,-178.673,6.911,148.893
C03137=1147.967,148.439,-57.914,-178.675,6.909,148.893
C03138=1147.972,148.189,-57.893,-178.678,6.907,148.894
C03139=1147.978,147.940,-57.872,-178.681,6.904,148.894
C03140=1147.982,147.691,-57.852,-178.684,6.903,148.894
C03141=1147.987,147.443,-57.830,-178.687,6.901,148.895
C03142=1147.991,147.194,-57.810,-178.690,6.899,148.895
C03143=1147.997,146.944,-57.789,-178.692,6.898,148.895
C03144=1148.001,146.695,-57.768,-178.696,6.895,148.896
C03145=1148.006,146.445,-57.747,-178.698,6.893,148.896
C03146=1148.010,146.197,-57.725,-178.701,6.892,148.897
C03147=1148.015,145.948,-57.705,-178.704,6.890,148.897
C03148=1148.020,145.699,-57.684,-178.706,6.888,148.897
C03149=1148.024,145.450,-57.664,-178.709,6.886,148.898
C03150=1148.030,145.200,-57.643,-178.712,6.884,148.898
C03151=1148.034,144.951,-57.622,-178.715,6.882,148.898
C03152=1148.039,144.702,-57.601,-178.717,6.880,148.899
C03153=1148.043,144.454,-57.580,-178.720,6.878,148.899
C03154=1148.049,144.205,-57.559,-178.723,6.877,148.899
C03155=1148.053,143.956,-57.539,-178.726,6.875,148.900
C03156=1148.058,143.706,-57.518,-178.729,6.872,148.900
C03157=1148.062,143.457,-57.497,-178.732,6.871,148.901
C03158=1148.067,143.207,-57.476,-178.734,6.869,148.901
C03159=1148.072,142.959,-57.456,-178.737,6.867,148.901
C03160=1148.076,142.710,-57.436,-178.740,6.866,148.902
C03161=1148.081,142.460,-57.415,-178.742,6.864,148.902
C03162=1148.086,142.211,-57.394,-178.745,6.861,148.902
C03163=1148.091,141.962,-57.373,-178.748,6.859,148.903
C03164=1148.095,141.713,-57.353,-178.751,6.858,148.903
C03165=1148.100,141.464,-57.332,-178.753,6.856,148.903
C03166=1148.105,141.215,-57.312,-178.756,6.854,148.904
C03167=1148.109,140.966,-57.291,-178.759,6.852,148.904
C03168=1148.114,140.717,-57.270,-178.761,6.851,148.905
C03169=1148.119,140.468,-57.250,-178.764,6.849,148.905
C03170=1148.124,140.218,-57.230,-178.768,6.847,148.905
C03171=1148.129,139.969,-57.209,-178.770,6.845,148.906
C03172=1148.133,139.720,-57.189,-178.773,6.843,148.906
C03173=1148.138,139.471,-57.168,-178.776,6.841,148.907
C03174=1148.143,139.222,-57.147,-178.778,6.840,148.907
C03175=1148.147,138.973,-57.127,-178.781,6.838,148.907
C03176=1148.152,138.724,-57.107,-178.784,6.836,148.908
C03177=1148.157,138.474,-57.086,-178.786,6.835,148.908
C03178=1148.162,138.226,-57.066,-178.790,6.832,148.908
C03179=1148.167,137.977,-57.046,-178.793,6.830,148.909
C03180=1148.172,137.728,-57.025,-178.795,6.829,148.909
C03181=1148.176,137.479,-57.005,-178.798,6.827,148.910
C03182=1148.181,137.229,-56.985,-178.801,6.825,148.910
C03183=1148.185,136.980,-56.965,-178.803,6.823,148.910
C03184=1148.191,136.731,-56.944,-178.806,6.822,148.911
C03185=1148.195,136.482,-56.923,-178.809,6.820,148.911
C03186=1148.200,136.232,-56.904,-178.812,6.818,148.912
C03187=1148.204,135.983,-56.883,-178.815,6.816,148.912
C03188=1148.209,135.734,-56.862,-178.818,6.814,148.912
C03189=1148.214,135.485,-56.843,-178.820,6.812,148.913
C03190=1148.219,135.236,-56.823,-178.823,6.811,148.913
C03191=1148.224,134.987,-56.802,-178.826,6.809,148.914
C03192=1148.229,134.737,-56.782,-178.828,6.807,148.914
C03193=1148.234,134.489,-56.762,-178.831,6.806,148.914
C03194=1148.238,134.240,-56.741,-178.834,6.804,148.915
C03195=1148.243,133.990,-56.722,-178.837,6.802,148.915
C03196=1148.247,133.741,-56.701,-178.839,6.800,148.916
C03197=1148.253,133.492,-56.682,-178.842,6.799,148.916
C03198=1148.258,133.243,-56.661,-178.845,6.797,148.916
C03199=1148.262,132.994,-56.641,-178.848,6.794,148.917
C03200=1148.267,132.744,-56.621,-178.851,6.793,148.917
C03201=1148.271,132.495,-56.601,-178.853,6.791,148.917
C03202=1148.276,132.246,-56.581,-178.856,6.789,148.918
C03203=1148.281,131.978,-56.559,-178.859,6.788,148.918
C03204=1148.286,131.709,-56.538,-178.862,6.786,148.919
C03205=1148.291,131.440,-56.516,-178.865,6.783,148.919
C03206=1148.297,131.173,-56.494,-178.868,6.782,148.919
C03207=1148.302,130.923,-56.475,-178.870,6.780,148.920
C03208=1148.306,130.674,-56.454,-178.873,6.778,148.920
C03209=1148.311,130.425,-56.435,-178.876,6.777,148.921
C03210=1148.316,130.175,-56.415,-178.879,6.775,148.921
C03211=1148.321,129.927,-56.395,-178.882,6.774,148.922
C03212=1148.326,129.677,-56.375,-178.884,6.772,148.922
C03213=1148.330,129.428,-56.355,-178.887,6.770,148.922
C03214=1148.335,129.179,-56.335,-178.890,6.768,148.923
C03215=1148.340,128.930,-56.316,-178.893,6.767,148.923
C03216=1148.345,128.681,-56.296,-178.895,6.765,148.924
C03217=1148.349,128.431,-56.276,-178.899,6.762,148.924
C03218=1148.354,128.182,-56.256,-178.901,6.761,148.924
C03219=1148.359,127.933,-56.236,-178.904,6.759,148.925
C03220=1148.364,127.684,-56.217,-178.907,6.757,148.925
C03221=1148.368,127.435,-56.196,-178.909,6.756,148.926
C03222=1148.373,127.185,-56.177,-178.912,6.754,148.926
C03223=1148.378,126.937,-56.157,-178.915,6.752,148.926
C03224=1148.383,126.687,-56.138,-178.918,6.751,148.927
C03225=1148.388,126.438,-56.117,-178.920,6.749,148.927
C03226=1148.393,126.189,-56.098,-178.923,6.747,148.928
C03227=1148.398,125.940,-56.078,-178.926,6.745,148.928
C03228=1148.402,125.691,-56.058,-178.928,6.744,148.928
C03229=1148.407,125.441,-56.038,-178.931,6.742,148.929
C03230=1148.412,125.192,-56.019,-178.934,6.740,148.929
C03231=1148.417,124.943,-55.999,-178.937,6.739,148.930
C03232=1148.421,124.693,-55.980,-178.939,6.737,148.930
C03233=1148.426,124.445,-55.960,-178.943,6.736,148.931
C03234=1148.431,124.196,-55.941,-178.945,6.734,148.931
C03235=1148.435,123.946,-55.921,-178.948,6.732,148.931
C03236=1148.441,123.697,-55.902,-178.951,6.730,148.932
C03237=1148.446,123.448,-55.882,-178.953,6.729,148.932
C03238=1148.450,123.198,-55.862,-178.956,6.727,148.933
C03239=1148.455,122.950,-55.843,-178.959,6.725,148.933
C03240=1148.459,122.700,-55.823,-178.962,6.724,148.933
C03241=1148.464,122.451,-55.804,-178.964,6.722,148.934
C03242=1148.469,122.202,-55.784,-178.967,6.720,148.934
C03243=1148.474,121.952,-55.765,-178.970,6.719,148.935
C03244=1148.480,121.704,-55.746,-178.972,6.717,148.935
C03245=1148.484,121.454,-55.726,-178.975,6.715,148.935
C03246=1148.488,121.205,-55.707,-178.978,6.714,148.936
C03247=1148.494,120.956,-55.688,-178.981,6.712,148.936
C03248=1148.498,120.706,-55.668,-178.984,6.710,148.937
C03249=1148.503,120.458,-55.649,-178.987,6.709,148.937
C03250=1148.508,120.208,-55.630,-178.989,6.707,148.938
C03251=1148.512,119.959,-55.610,-178.992,6.705,148.938
C03252=1148.518,119.710,-55.591,-178.995,6.704,148.938
C03253=1148.522,119.460,-55.572,-178.997,6.702,148.939
C03254=1148.527,119.212,-55.552,-179.000,6.700,148.939
C03255=1148.532,118.962,-55.533,-179.003,6.699,148.940
C03256=1148.537,118.713,-55.513,-179.006,6.697,148.940
C03257=1148.541,118.464,-55.494,-179.009,6.695,148.941
C03258=1148.546,118.214,-55.475,-179.011,6.694,148.941
C03259=1148.551,117.966,-55.455,-179.014,6.693,148.941
C03260=1148.555,117.716,-55.436,-179.016,6.691,148.942
C03261=1148.561,117.467,-55.418,-179.019,6.689,148.942
C03262=1148.566,117.217,-55.398,-179.022,6.688,148.943
C03263=1148.570,116.969,-55.379,-179.025,6.686,148.943
C03264=1148.575,116.719,-55.360,-179.027,6.684,148.944
C03265=1148.580,116.470,-55.340,-179.030,6.683,148.944
C03266=1148.584,116.221,-55.321,-179.033,6.681,148.944
C03267=1148.590,115.971,-55.303,-179.036,6.680,148.945
C03268=1148.595,115.722,-55.283,-179.039,6.678,148.945
C03269=1148.599,115.473,-55.264,-179.041,6.676,148.946
C03270=1148.604,115.224,-55.245,-179.044,6.675,148.946
C03271=1148.609,114.975,-55.226,-179.047,6.673,148.947
C03272=1148.614,114.725,-55.207,-179.050,6.671,148.947
C03273=1148.619,114.476,-55.188,-179.052,6.669,148.947
C03274=1148.623,114.227,-55.169,-179.055,6.668,148.948
C03275=1148.629,113.978,-55.149,-179.058,6.666,148.948
C03276=1148.633,113.728,-55.131,-179.061,6.665,148.949
C03277=1148.638,113.479,-55.112,-179.063,6.664,148.949
C03278=1148.643,113.231,-55.093,-179.066,6.662,148.950
C03279=1148.648,112.981,-55.074,-179.068,6.660,148.950
C03280=1148.653,112.732,-55.055,-179.071,6.659,148.950
C03281=1148.657,112.482,-55.036,-179.074,6.657,148.951
C03282=1148.663,112.233,-55.017,-179.077,6.655,148.951
C03283=1148.667,111.984,-54.998,-179.080,6.654,148.952
C03284=1148.672,111.735,-54.979,-179.083,6.652,148.952
C03285=1148.677,111.486,-54.961,-179.085,6.651,148.953
C03286=1148.682,111.236,-54.941,-179.088,6.649,148.953
C03287=1148.687,110.987,-54.923,-179.091,6.647,148.954
C03288=1148.691,110.737,-54.904,-179.093,6.646,148.954
C03289=1148.696,110.489,-54.885,-179.096,6.645,148.954
C03290=1148.701,110.240,-54.867,-179.099,6.643,148.955
C03291=1148.706,109.990,-54.847,-179.102,6.642,148.955
C03292=1148.711,109.741,-54.829,-179.104,6.640,148.956
C03293=1148.715,109.491,-54.810,-179.107,6.638,148.956
C03294=1148.720,109.242,-54.792,-179.110,6.637,148.957
C03295=1148.726,108.993,-54.772,-179.112,6.635,148.957
C03296=1148.730,108.743,-54.754,-179.116,6.634,148.958
C03297=1148.735,108.495,-54.735,-179.118,6.632,148.958
C03298=1148.740,108.245,-54.717,-179.121,6.630,148.958
C03299=1148.744,107.996,-54.698,-179.123,6.629,148.959
C03300=1148.750,107.747,-54.679,-179.126,6.628,148.959
C03301=1148.754,107.497,-54.660,-179.129,6.626,148.960
C03302=1148.759,107.248,-54.642,-179.131,6.624,148.960
C03303=1148.764,106.999,-54.623,-179.135,6.623,148.961
C03304=1148.768,106.749,-54.604,-179.137,6.621,148.961
C03305=1148.773,106.500,-54.586,-179.140,6.620,148.962
C03306=1148.779,106.251,-54.567,-179.143,6.618,148.962
C03307=1148.784,105.983,-54.548,-179.146,6.616,148.962
C03308=1148.789,105.714,-54.527,-179.149,6.615,148.963
C03309=1148.794,105.446,-54.507,-179.151,6.613,148.963
C03310=1148.800,105.178,-54.487,-179.155,6.612,148.964
C03311=1148.805,104.928,-54.469,-179.157,6.610,148.964
C03312=1148.809,104.679,-54.450,-179.160,6.608,148.965
C03313=1148.814,104.430,-54.432,-179.163,6.607,148.965
C03314=1148.819,104.181,-54.414,-179.165,6.606,148.966
C03315=1148.824,103.931,-54.396,-179.168,6.604,148.966
C03316=1148.828,103.682,-54.377,-179.171,6.603,148.967
C03317=1148.834,103.433,-54.358,-179.174,6.601,148.967
C03318=1148.839,103.183,-54.340,-179.176,6.599,148.968
C03319=1148.843,102.934,-54.321,-179.179,6.598,148.968
C03320=1148.847,102.685,-54.303,-179.181,6.597,148.968
C03321=1148.853,102.436,-54.284,-179.184,6.596,148.969
C03322=1148.858,102.186,-54.266,-179.187,6.594,148.969
C03323=1148.862,101.936,-54.248,-179.190,6.592,148.970
C03324=1148.867,101.688,-54.229,-179.193,6.590,148.970
C03325=1148.872,101.439,-54.211,-179.195,6.589,148.971
C03326=1148.878,101.189,-54.193,-179.198,6.587,148.971
C03327=1148.882,100.940,-54.175,-179.201,6.587,148.972
C03328=1148.887,100.690,-54.157,-179.203,6.585,148.972
C03329=1148.892,100.441,-54.139,-179.206,6.583,148.973
C03330=1148.896,100.192,-54.120,-179.209,6.582,148.973
C03331=1148.902,99.943,-54.101,-179.212,6.580,148.973
C03332=1148.907,99.694,-54.083,-179.214,6.579,148.974
C03333=1148.911,99.444,-54.065,-179.217,6.578,148.974
C03334=1148.916,99.195,-54.047,-179.220,6.576,148.975
C03335=1148.921,98.946,-54.029,-179.222,6.574,148.975
C03336=1148.926,98.696,-54.011,-179.226,6.573,148.976
C03337=1148.931,98.447,-53.993,-179.228,6.571,148.976
C03338=1148.936,98.198,-53.975,-179.231,6.570,148.977
C03339=1148.940,97.948,-53.957,-179.233,6.569,148.977
C03340=1148.946,97.699,-53.938,-179.236,6.567,148.978
C03341=1148.951,97.449,-53.920,-179.239,6.566,148.978
C03342=1148.955,97.200,-53.902,-179.242,6.564,148.979
C03343=1148.960,96.951,-53.884,-179.244,6.563,148.979
C03344=1148.965,96.702,-53.866,-179.247,6.561,148.980
C03345=1148.970,96.452,-53.848,-179.250,6.560,148.980
C03346=1148.975,96.203,-53.830,-179.253,6.558,148.981
C03347=1148.979,95.954,-53.812,-179.256,6.557,148.981
C03348=1148.984,95.705,-53.794,-179.258,6.556,148.981
C03349=1148.989,95.455,-53.776,-179.260,6.554,148.982
C03350=1148.994,95.206,-53.758,-179.264,6.553,148.982
C03351=1148.999,94.957,-53.740,-179.266,6.551,148.983
C03352=1149.004,94.708,-53.722,-179.269,6.550,148.983
C03353=1149.009,94.459,-53.704,-179.271,6.549,148.984
C03354=1149.013,94.209,-53.686,-179.274,6.547,148.984
C03355=1149.018,93.960,-53.668,-179.277,6.546,148.985
C03356=1149.023,93.710,-53.650,-179.280,6.544,148.985
C03357=1149.028,93.461,-53.632,-179.283,6.542,148.986
C03358=1149.033,93.211,-53.614,-179.285,6.541,148.986
C03359=1149.038,92.962,-53.597,-179.288,6.540,148.987
C03360=1149.043,92.713,-53.579,-179.291,6.538,148.987
C03361=1149.048,92.464,-53.561,-179.293,6.537,148.988
C03362=1149.053,92.214,-53.543,-179.296,6.536,148.988
C03363=1149.058,91.965,-53.525,-179.299,6.535,148.989
C03364=1149.063,91.716,-53.507,-179.302,6.533,148.989
C03365=1149.068,91.467,-53.489,-179.304,6.531,148.989
C03366=1149.072,91.217,-53.473,-179.306,6.530,148.990
C03367=1149.077,90.968,-53.455,-179.310,6.529,148.990
C03368=1149.082,90.719,-53.437,-179.312,6.527,148.991
C03369=1149.087,90.470,-53.419,-179.315,6.526,148.991
C03370=1149.092,90.220,-53.401,-179.317,6.525,148.992
C03371=1149.097,89.971,-53.383,-179.320,6.523,148.992
C03372=1149.102,89.721,-53.366,-179.323,6.522,148.993
C03373=1149.107,89.472,-53.348,-179.326,6.520,148.993
C03374=1149.112,89.223,-53.331,-179.328,6.519,148.994
C03375=1149.116,88.974,-53.313,-179.331,6.518,148.994
C03376=1149.122,88.724,-53.296,-179.334,6.516,148.995
C03377=1149.127,88.475,-53.278,-179.337,6.515,148.995
C03378=1149.131,88.226,-53.260,-179.339,6.514,148.996
C03379=1149.136,87.976,-53.243,-179.342,6.512,148.996
C03380=1149.141,87.727,-53.225,-179.345,6.511,148.997
C03381=1149.146,87.478,-53.207,-179.348,6.509,148.997
C03382=1149.151,87.228,-53.190,-179.350,6.508,148.998
C03383=1149.156,86.979,-53.172,-179.353,6.507,148.998
C03384=1149.160,86.729,-53.155,-179.356,6.505,148.999
C03385=1149.165,86.480,-53.137,-179.358,6.503,148.999
C03386=1149.171,86.230,-53.120,-179.361,6.503,148.999
C03387=1149.175,85.981,-53.102,-179.364,6.501,149.000
C03388=1149.180,85.732,-53.085,-179.367,6.500,149.000
C03389=1149.185,85.482,-53.067,-179.369,6.499,149.001
C03390=1149.190,85.233,-53.050,-179.372,6.497,149.002
C03391=1149.195,84.983,-53.032,-179.375,6.496,149.002
C03392=1149.199,84.734,-53.015,-179.377,6.494,149.002
C03393=1149.205,84.485,-52.998,-179.379,6.493,149.003
C03394=1149.210,84.236,-52.980,-179.383,6.492,149.003
C03395=1149.214,83.987,-52.963,-179.385,6.490,149.004
C03396=1149.220,83.737,-52.946,-179.388,6.489,149.004
C03397=1149.224,83.488,-52.928,-179.390,6.488,149.005
C03398=1149.230,83.238,-52.911,-179.394,6.486,149.005
C03399=1149.234,82.989,-52.893,-179.396,6.485,149.006
C03400=1149.239,82.739,-52.876,-179.398,6.484,149.006
C03401=1149.244,82.490,-52.859,-179.402,6.483,149.007
C03402=1149.249,82.241,-52.842,-179.404,6.481,149.007
C03403=1149.254,81.992,-52.824,-179.407,6.480,149.008
C03404=1149.258,81.743,-52.807,-179.409,6.478,149.008
C03405=1149.264,81.493,-52.790,-179.412,6.477,149.009
C03406=1149.269,81.243,-52.772,-179.415,6.476,149.009
C03407=1149.273,80.994,-52.755,-179.417,6.474,149.010
C03408=1149.278,80.745,-52.738,-179.421,6.473,149.010
C03409=1149.284,80.495,-52.721,-179.423,6.471,149.011
C03410=1149.288,80.247,-52.704,-179.425,6.471,149.011
C03411=1149.294,79.978,-52.685,-179.429,6.469,149.012
C03412=1149.299,79.710,-52.667,-179.431,6.468,149.012
C03413=1149.304,79.441,-52.648,-179.435,6.466,149.013
C03414=1149.310,79.172,-52.630,-179.437,6.465,149.013
C03415=1149.315,78.923,-52.613,-179.440,6.464,149.014
C03416=1149.320,78.674,-52.595,-179.443,6.463,149.014
C03417=1149.324,78.425,-52.579,-179.446,6.461,149.015
C03418=1149.329,78.175,-52.561,-179.448,6.460,149.015
C03419=1149.334,77.925,-52.545,-179.451,6.459,149.016
C03420=1149.340,77.676,-52.528,-179.454,6.457,149.016
C03421=1149.344,77.427,-52.511,-179.456,6.456,149.017
C03422=1149.349,77.178,-52.493,-179.459,6.454,149.017
C03423=1149.354,76.928,-52.477,-179.462,6.453,149.018
C03424=1149.359,76.678,-52.459,-179.464,6.452,149.018
C03425=1149.364,76.430,-52.443,-179.467,6.451,149.019
C03426=1149.369,76.180,-52.426,-179.470,6.449,149.019
C03427=1149.373,75.931,-52.408,-179.472,6.448,149.020
C03428=1149.378,75.681,-52.391,-179.475,6.447,149.020
C03429=1149.384,75.432,-52.375,-179.478,6.445,149.021
C03430=1149.389,75.183,-52.358,-179.480,6.445,149.021
C03431=1149.393,74.933,-52.341,-179.483,6.443,149.022
C03432=1149.399,74.684,-52.324,-179.486,6.442,149.022
C03433=1149.404,74.434,-52.307,-179.488,6.441,149.023
C03434=1149.408,74.185,-52.291,-179.491,6.439,149.023
C03435=1149.413,73.935,-52.273,-179.494,6.438,149.024
C03436=1149.418,73.686,-52.257,-179.496,6.437,149.024
C03437=1149.424,73.437,-52.240,-179.499,6.435,149.025
C03438=1149.428,73.187,-52.223,-179.501,6.434,149.025
C03439=1149.433,72.938,-52.207,-179.504,6.433,149.026
C03440=1149.438,72.689,-52.190,-179.507,6.431,149.026
C03441=1149.443,72.439,-52.173,-179.509,6.431,149.027
C03442=1149.448,72.189,-52.156,-179.513,6.429,149.027
C03443=1149.453,71.940,-52.139,-179.515,6.428,149.028
C03444=1149.458,71.691,-52.123,-179.517,6.427,149.028
C03445=1149.463,71.441,-52.105,-179.521,6.425,149.029
C03446=1149.468,71.192,-52.089,-179.523,6.425,149.029
C03447=1149.472,70.943,-52.072,-179.526,6.423,149.030
C03448=1149.478,70.693,-52.055,-179.529,6.422,149.030
C03449=1149.483,70.444,-52.039,-179.531,6.421,149.031
C03450=1149.487,70.195,-52.022,-179.534,6.419,149.031
C03451=1149.493,69.946,-52.005,-179.537,6.418,149.032
C03452=1149.497,69.696,-51.989,-179.539,6.417,149.032
C03453=1149.502,69.446,-51.973,-179.542,6.415,149.033
C03454=1149.507,69.197,-51.956,-179.544,6.415,149.034
C03455=1149.513,68.948,-51.939,-179.547,6.413,149.034
C03456=1149.517,68.698,-51.922,-179.550,6.411,149.034
C03457=1149.522,68.449,-51.906,-179.553,6.411,149.035
C03458=1149.527,68.200,-51.889,-179.555,6.409,149.035
C03459=1149.533,67.950,-51.873,-179.557,6.408,149.036
C03460=1149.537,67.701,-51.857,-179.561,6.407,149.037
C03461=1149.542,67.451,-51.840,-179.563,6.406,149.037
C03462=1149.547,67.202,-51.824,-179.566,6.405,149.037
C03463=1149.552,66.953,-51.806,-179.569,6.403,149.038
C03464=1149.557,66.703,-51.791,-179.571,6.402,149.039
C03465=1149.562,66.454,-51.774,-179.574,6.401,149.039
C03466=1149.566,66.204,-51.757,-179.576,6.400,149.040
C03467=1149.571,65.955,-51.741,-179.579,6.399,149.040
C03468=1149.577,65.705,-51.725,-179.582,6.397,149.041
C03469=1149.582,65.456,-51.708,-179.584,6.397,149.041
C03470=1149.586,65.207,-51.692,-179.587,6.395,149.042
C03471=1149.592,64.957,-51.676,-179.590,6.394,149.042
C03472=1149.596,64.708,-51.659,-179.593,6.393,149.043
C03473=1149.601,64.458,-51.643,-179.595,6.392,149.043
C03474=1149.607,64.209,-51.627,-179.598,6.391,149.044
C03475=1149.611,63.959,-51.610,-179.601,6.389,149.044
C03476=1149.616,63.710,-51.594,-179.603,6.388,149.045
C03477=1149.621,63.460,-51.578,-179.606,6.387,149.045
C03478=1149.626,63.212,-51.561,-179.608,6.386,149.046
C03479=1149.631,62.962,-51.545,-179.611,6.384,149.046
C03480=1149.636,62.713,-51.529,-179.614,6.384,149.047
C03481=1149.641,62.463,-51.512,-179.616,6.382,149.047
C03482=1149.646,62.214,-51.497,-179.620,6.381,149.048
C03483=1149.651,61.964,-51.480,-179.622,6.380,149.048
C03484=1149.656,61.715,-51.463,-179.624,6.378,149.049
C03485=1149.661,61.465,-51.447,-179.627,6.378,149.049
C03486=1149.666,61.216,-51.431,-179.630,6.376,149.050
C03487=1149.671,60.966,-51.415,-179.632,6.375,149.050
C03488=1149.676,60.717,-51.399,-179.635,6.374,149.051
C03489=1149.681,60.467,-51.383,-179.637,6.373,149.051
C03490=1149.686,60.219,-51.366,-179.640,6.371,149.052
C03491=1149.691,59.968,-51.350,-179.643,6.371,149.053
C03492=1149.696,59.720,-51.334,-179.646,6.369,149.053
C03493=1149.701,59.470,-51.319,-179.649,6.368,149.054
C03494=1149.706,59.221,-51.302,-179.651,6.367,149.054
C03495=1149.711,58.971,-51.286,-179.654,6.366,149.055
C03496=1149.716,58.722,-51.270,-179.656,6.365,149.055
C03497=1149.721,58.472,-51.254,-179.659,6.363,149.056
C03498=1149.726,58.222,-51.238,-179.661,6.363,149.056
C03499=1149.731,57.974,-51.222,-179.664,6.361,149.057
C03500=1149.736,57.724,-51.206,-179.667,6.360,149.057
C03501=1149.741,57.475,-51.190,-179.669,6.359,149.058
C03502=1149.746,57.225,-51.174,-179.672,6.358,149.058
C03503=1149.751,56.975,-51.158,-179.675,6.357,149.059
C03504=1149.756,56.726,-51.142,-179.677,6.356,149.059
C03505=1149.761,56.476,-51.126,-179.680,6.354,149.060
C03506=1149.766,56.227,-51.110,-179.682,6.354,149.060
C03507=1149.771,55.978,-51.094,-179.686,6.352,149.061
C03508=1149.776,55.728,-51.078,-179.688,6.352,149.061
C03509=1149.781,55.479,-51.063,-179.691,6.350,149.062
C03510=1149.786,55.230,-51.047,-179.693,6.349,149.062
C03511=1149.791,54.980,-51.031,-179.696,6.348,149.063
C03512=1149.796,54.731,-51.015,-179.698,6.347,149.064
C03513=1149.800,54.481,-50.998,-179.701,6.346,149.064
C03514=1149.806,54.232,-50.983,-179.703,6.345,149.064
C03515=1149.811,53.963,-50.966,-179.707,6.343,149.065
C03516=1149.817,53.695,-50.949,-179.710,6.342,149.066
C03517=1149.822,53.426,-50.932,-179.712,6.341,149.066
C03518=1149.827,53.157,-50.914,-179.715,6.340,149.067
C03519=1149.832,52.908,-50.899,-179.718,6.338,149.067
C03520=1149.837,52.659,-50.884,-179.720,6.338,149.068
C03521=1149.842,52.409,-50.868,-179.723,6.336,149.068
C03522=1149.847,52.160,-50.852,-179.725,6.335,149.069
C03523=1149.853,51.910,-50.836,-179.729,6.334,149.070
C03524=1149.857,51.660,-50.820,-179.731,6.333,149.070
C03525=1149.862,51.411,-50.805,-179.734,6.332,149.070
C03526=1149.868,51.162,-50.789,-179.736,6.331,149.071
C03527=1149.872,50.912,-50.773,-179.738,6.330,149.072
C03528=1149.877,50.663,-50.757,-179.742,6.329,149.072
C03529=1149.882,50.414,-50.742,-179.744,6.328,149.073
C03530=1149.887,50.164,-50.727,-179.747,6.327,149.073
C03531=1149.892,49.914,-50.711,-179.749,6.326,149.074
C03532=1149.898,49.665,-50.695,-179.752,6.324,149.074
C03533=1149.902,49.416,-50.680,-179.755,6.324,149.075
C03534=1149.907,49.166,-50.664,-179.757,6.322,149.075
C03535=1149.912,48.916,-50.649,-179.760,6.321,149.076
C03536=1149.918,48.667,-50.633,-179.763,6.320,149.076
C03537=1149.922,48.418,-50.618,-179.765,6.319,149.077
C03538=1149.927,48.168,-50.602,-179.768,6.318,149.078
C03539=1149.933,47.918,-50.586,-179.770,6.317,149.078
C03540=1149.938,47.669,-50.571,-179.773,6.316,149.078
C03541=1149.943,47.420,-50.556,-179.776,6.315,149.079
C03542=1149.947,47.170,-50.540,-179.778,6.314,149.080
C03543=1149.953,46.920,-50.524,-179.781,6.313,149.080
C03544=1149.957,46.671,-50.509,-179.783,6.312,149.081
C03545=1149.963,46.422,-50.494,-179.786,6.310,149.081
C03546=1149.968,46.172,-50.478,-179.789,6.310,149.082
C03547=1149.972,45.923,-50.463,-179.791,6.308,149.082
C03548=1149.978,45.673,-50.447,-179.794,6.308,149.083
C03549=1149.982,45.424,-50.432,-179.797,6.306,149.083
C03550=1149.988,45.175,-50.417,-179.799,6.305,149.084
C03551=1149.993,44.925,-50.401,-179.802,6.305,149.084
C03552=1149.997,44.675,-50.386,-179.804,6.303,149.085
C03553=1150.003,44.426,-50.370,-179.807,6.303,149.086
C03554=1150.008,44.177,-50.354,-179.810,6.301,149.086
C03555=1150.013,43.928,-50.339,-179.812,6.301,149.087
C03556=1150.018,43.678,-50.324,-179.815,6.299,149.087
C03557=1150.022,43.428,-50.309,-179.817,6.298,149.088
C03558=1150.028,43.178,-50.294,-179.820,6.298,149.088
C03559=1150.033,42.929,-50.278,-179.823,6.296,149.089
C03560=1150.038,42.680,-50.263,-179.825,6.296,149.089
C03561=1150.043,42.430,-50.247,-179.828,6.294,149.090
C03562=1150.048,42.181,-50.232,-179.830,6.293,149.090
C03563=1150.053,41.931,-50.217,-179.833,6.292,149.091
C03564=1150.058,41.682,-50.202,-179.836,6.291,149.091
C03565=1150.063,41.432,-50.187,-179.838,6.290,149.092
C03566=1150.068,41.183,-50.172,-179.841,6.289,149.093
C03567=1150.073,40.933,-50.157,-179.844,6.288,149.093
C03568=1150.078,40.684,-50.142,-179.846,6.287,149.094
C03569=1150.083,40.435,-50.126,-179.849,6.286,149.094
C03570=1150.088,40.185,-50.111,-179.851,6.285,149.095
C03571=1150.094,39.935,-50.096,-179.854,6.284,149.095
C03572=1150.098,39.686,-50.081,-179.857,6.283,149.096
C03573=1150.103,39.436,-50.065,-179.859,6.282,149.096
C03574=1150.108,39.187,-50.050,-179.862,6.281,149.097
C03575=1150.113,38.937,-50.036,-179.864,6.280,149.097
C03576=1150.118,38.688,-50.021,-179.867,6.279,149.098
C03577=1150.123,38.439,-50.005,-179.870,6.278,149.099
C03578=1150.128,38.189,-49.991,-179.872,6.277,149.099
C03579=1150.134,37.940,-49.975,-179.875,6.276,149.100
C03580=1150.138,37.690,-49.960,-179.877,6.275,149.100
C03581=1150.144,37.440,-49.945,-179.880,6.274,149.101
C03582=1150.149,37.191,-49.930,-179.883,6.273,149.101
C03583=1150.154,36.941,-49.915,-179.885,6.272,149.102
C03584=1150.159,36.692,-49.900,-179.888,6.271,149.102
C03585=1150.163,36.442,-49.885,-179.890,6.270,149.103
C03586=1150.169,36.192,-49.870,-179.893,6.269,149.104
C03587=1150.174,35.943,-49.855,-179.896,6.268,149.104
C03588=1150.179,35.693,-49.840,-179.898,6.267,149.104
C03589=1150.184,35.444,-49.825,-179.901,6.266,149.105
C03590=1150.189,35.194,-49.811,-179.903,6.265,149.106
C03591=1150.194,34.945,-49.795,-179.906,6.265,149.106
C03592=1150.199,34.696,-49.780,-179.909,6.263,149.107
C03593=1150.204,34.446,-49.766,-179.911,6.263,149.107
C03594=1150.209,34.197,-49.751,-179.914,6.261,149.108
C03595=1150.214,33.947,-49.736,-179.916,6.260,149.108
C03596=1150.219,33.698,-49.721,-179.919,6.260,149.109
C03597=1150.224,33.448,-49.706,-179.921,6.258,149.109
C03598=1150.229,33.199,-49.691,-179.924,6.258,149.110
C03599=1150.234,32.949,-49.677,-179.926,6.257,149.110
C03600=1150.240,32.699,-49.662,-179.930,6.255,149.111
C03601=1150.244,32.450,-49.647,-179.932,6.255,149.112
C03602=1150.249,32.200,-49.633,-179.934,6.254,149.112
C03603=1150.255,31.951,-49.617,-179.937,6.253,149.113
C03604=1150.260,31.701,-49.603,-179.939,6.252,149.113
C03605=1150.264,31.452,-49.588,-179.942,6.251,149.114
C03606=1150.269,31.202,-49.574,-179.945,6.250,149.114
C03607=1150.276,30.953,-49.559,-179.947,6.249,149.115
C03608=1150.280,30.704,-49.544,-179.950,6.248,149.115
C03609=1150.285,30.454,-49.530,-179.953,6.247,149.116
C03610=1150.290,30.205,-49.515,-179.955,6.246,149.117
C03611=1150.296,29.955,-49.500,-179.958,6.245,149.117
C03612=1150.301,29.706,-49.486,-179.960,6.244,149.118
C03613=1150.305,29.456,-49.471,-179.962,6.243,149.118
C03614=1150.310,29.207,-49.457,-179.966,6.242,149.119
C03615=1150.316,28.957,-49.442,-179.968,6.241,149.119
C03616=1150.320,28.708,-49.427,-179.970,6.241,149.120
C03617=1150.325,28.458,-49.413,-179.973,6.240,149.120
C03618=1150.330,28.208,-49.398,-179.976,6.239,149.121
C03619=1150.335,27.939,-49.383,-179.978,6.238,149.122
C03620=1150.342,27.671,-49.367,-179.981,6.237,149.122
C03621=1150.347,27.402,-49.351,-179.983,6.236,149.123
C03622=1150.353,27.133,-49.336,-179.987,6.234,149.123
C03623=1150.357,26.884,-49.321,-179.989,6.234,149.124
C03624=1150.363,26.634,-49.306,-179.992,6.233,149.125
C03625=1150.368,26.384,-49.292,-179.994,6.232,149.125
C03626=1150.373,26.134,-49.278,-179.997,6.231,149.126
C03627=1150.378,25.885,-49.263,-179.999,6.230,149.126
C03628=1150.382,25.635,-49.248,179.998,6.229,149.127
C03629=1150.388,25.386,-49.234,179.995,6.228,149.127
C03630=1150.393,25.137,-49.220,179.993,6.228,149.128
C03631=1150.399,24.887,-49.205,179.990,6.226,149.128
C03632=1150.404,24.637,-49.191,179.987,6.226,149.129
C03633=1150.408,24.388,-49.176,179.985,6.225,149.129
C03634=1150.413,24.138,-49.162,179.982,6.223,149.130
C03635=1150.419,23.889,-49.148,179.980,6.223,149.131
C03636=1150.424,23.640,-49.133,179.978,6.222,149.131
C03637=1150.429,23.390,-49.119,179.975,6.221,149.132
C03638=1150.434,23.140,-49.105,179.972,6.220,149.132
C03639=1150.439,22.890,-49.091,179.970,6.219,149.133
C03640=1150.443,22.641,-49.076,179.967,6.218,149.133
C03641=1150.449,22.392,-49.062,179.964,6.217,149.134
C03642=1150.454,22.143,-49.047,179.962,6.216,149.134
C03643=1150.459,21.893,-49.033,179.959,6.216,149.135
C03644=1150.464,21.643,-49.019,179.957,6.215,149.136
C03645=1150.469,21.393,-49.005,179.954,6.213,149.136
C03646=1150.474,21.144,-48.991,179.952,6.213,149.137
C03647=1150.479,20.895,-48.976,179.950,6.212,149.137
C03648=1150.484,20.645,-48.962,179.946,6.211,149.138
